   IF #command > 100 THEN
       "SandBoxData".MnualCommandMem := #command;
   END_IF;
   IF #command = 5000 THEN
       #data.Status.ToBp := true;
   END_IF;
   IF #command = 6000 THEN
       #data.Status.ToWp := true;
   END_IF;
   IF #command = 7000 THEN
       #data.Status.ToFp := true;
   END_IF;
END_REGION

REGION Network 3 (SCL): check new cylinder command
   //check if basic position req movement changed
   IF #data.Status.ToBp <> #dataOld.Status.ToBp AND #data.Status.ToBp THEN
       #data.Status.ToFp := false;
       #data.Status.ToWp := false;
       IF #noCollision THEN
           #data.Status.ToFp := false;
           #data.Status.ToWp := false;
       ELSE
           #data.Status.ToBp := false;
       END_IF;
   END_IF;
   //check if work position req movement changed
   IF #data.Status.ToWp <> #dataOld.Status.ToWp AND #data.Status.ToWp THEN
       IF #noCollision  THEN
           #data.Status.ToFp := false;
           #data.Status.ToBp := false;
       ELSE
           #data.Status.ToWp := false;
       END_IF;
   END_IF;
   //check if free position req movement changed
   IF #data.Status.ToFp <> #dataOld.Status.ToFp AND #data.Status.ToFp THEN
       #data.Status.ToBp := false;
       #data.Status.ToWp := false;
       IF #noCollision THEN
           #data.Status.ToBp := false;
           #data.Status.ToWp := false;
       ELSE
           #data.Status.ToFp := false;
       END_IF;
   END_IF;
   //store actual cylinder status to old
   #dataOld.Status := #data.Status;
END_REGION

REGION Network 4
   RUNG wire#powerrail
      Contact( #HydraulicActive )
      { S7_Templates := "time_type := Time" } #IEC_Timer_0_Instance.TON(pt := t#3s, et =>)
   END_RUNG
   // the same network as SCL:
   #IEC_Timer_0_Instance(IN := #HydraulicActive, PT := t#3s);   // TON
END_REGION

REGION Network 5: Start move to basic position
   RUNG wire#powerrail
      Contact( #data.Status.ToBp )
      Contact( #IEC_Timer_0_Instance.Q )
      Sub(in1 := 0.0, in2 := #data.FlowCmd, out => #data.Flow)
      Move(in := #data.PressureCmd, out1 => #data.Pressure)
   END_RUNG
   // the same network as SCL:
   IF #data.Status.ToBp AND #IEC_Timer_0_Instance.Q THEN
       #data.Flow := 0.0 - #data.FlowCmd;
       #data.Pressure := #data.PressureCmd;
   END_IF;
END_REGION

REGION Network 6: Start move to working position
   RUNG wire#powerrail
      Contact( #data.Status.ToWp )
      Contact( #IEC_Timer_0_Instance.Q )
      Move(in := #data.FlowCmd, out1 => #data.Flow)
      Move(in := #data.PressureCmd, out1 => #data.Pressure)
   END_RUNG
   // the same network as SCL:
   IF #data.Status.ToWp AND #IEC_Timer_0_Instance.Q THEN
       #data.Flow := #data.FlowCmd;
       #data.Pressure := #data.PressureCmd;
   END_IF;
END_REGION

REGION Network 7: Small movement to basic position when no command active and hydraulic running
   RUNG wire#powerrail
      Contact( #HydraulicActive )
      I_Contact( #data.Status.ToBp )
      I_Contact( #data.Status.ToWp )
      I_Contact( #data.Status.ToFp )
      { S7_Templates := "SrcType := Real" } LE_Contact(in1 := #data.Position, in2 := #BasicPositionMax)
      { S7_Templates := "SrcType := Real" } GE_Contact(in1 := #data.Position, in2 := #BasicPositionMin)
      Move(in := 3.0, out1 => #data.Pressure)
      Move(in := -5.0, out1 => #data.Flow)
   END_RUNG
   // the same network as SCL:
   IF #HydraulicActive AND NOT #data.Status.ToBp AND NOT #data.Status.ToWp AND NOT #data.Status.ToFp AND (#data.Position <= #BasicPositionMax) AND (#data.Position >= #BasicPositionMin) THEN
       #data.Pressure := 3.0;
       #data.Flow := -5.0;
   END_IF;
END_REGION

REGION Network 8: Stop movement when abou allowed position
   RUNG wire#powerrail
      { S7_Templates := "SrcType := Real" } GT_Contact(in1 := #data.Position, in2 := #MaxPosition)
      wire#w1
      I_Contact( #data.Status.ToBp )
      Contact( #HydraulicActive )
      Move(in := 3.0, out1 => #data.Pressure)
      Move(in := -5.0, out1 => #data.Flow)
   END_RUNG
   RUNG wire#w1
      I_Contact( #data.Status.ToBp )
      I_Contact( #HydraulicActive )
      Move(in := 0.0, out1 => #data.Pressure)
      Move(in := 0.0, out1 => #data.Flow)
   END_RUNG
   // the same network as SCL:
   #_w1 := #data.Position > #MaxPosition;
   IF #_w1 AND NOT #data.Status.ToBp AND #HydraulicActive THEN
       #data.Pressure := 3.0;
       #data.Flow := -5.0;
   END_IF;
   IF #_w1 AND NOT #data.Status.ToBp AND NOT #HydraulicActive THEN
       #data.Pressure := 0.0;
       #data.Flow := 0.0;
   END_IF;
END_REGION

REGION Network 9: In basic position
   RUNG wire#powerrail
      Contact( #data.Status.ToBp )
      wire#w1
      I_Contact( "FirstScan" )
      wire#w2
      Add(in1 := #BasicPositionMin, in2 := 1.0, out => #BasicPositionMin_1mm_margin)
      Add(in1 := #BasicPositionMax, in2 := -1.0, out => #BasicPositionMax_1mm_margin)
   END_RUNG
   RUNG wire#powerrail
      Contact( #data.Status.ToFp )
   END_RUNG wire#w1
   RUNG wire#w2
      { S7_Templates := "SrcType := Real" } GE_Contact(in1 := #data.Position, in2 := #BasicPositionMin)
      { S7_Templates := "SrcType := Real" } LE_Contact(in1 := #data.Position, in2 := #BasicPositionMax)
      { S7_Templates := "time_type := Time" } #IEC_Timer_0_Instance_1.TON(pt := t#50ms, et =>)
   END_RUNG
   RUNG wire#w2
      { S7_Templates := "SrcType := Real" } GE_Contact(in1 := #data.Position, in2 := #BasicPositionMin_1mm_margin)
      { S7_Templates := "SrcType := Real" } LE_Contact(in1 := #data.Position, in2 := #BasicPositionMax_1mm_margin)
      Coil( #data.InBp_1mm_margin )
   END_RUNG
   RUNG wire#w2
      Contact( #IEC_Timer_0_Instance_1.Q )
      wire#w3
      Coil( #data.Status.InBp )
   END_RUNG
   RUNG wire#w2
      Contact( #data.InBp_1mm_margin )
   END_RUNG wire#w3
   // the same network as SCL:
   #_w1 := (#data.Status.ToBp OR #data.Status.ToFp) AND NOT "FirstScan";
   IF #_w1 THEN
       #BasicPositionMin_1mm_margin := #BasicPositionMin + 1.0;
       #BasicPositionMax_1mm_margin := #BasicPositionMax + (-1.0);
   END_IF;
   #IEC_Timer_0_Instance_1(IN := #_w1 AND (#data.Position >= #BasicPositionMin) AND (#data.Position <= #BasicPositionMax),   // TON
                           PT := t#50ms);
   #data.InBp_1mm_margin := #_w1 AND (#data.Position >= #BasicPositionMin_1mm_margin) AND (#data.Position <= #BasicPositionMax_1mm_margin);
   #data.Status.InBp := #_w1 AND (#IEC_Timer_0_Instance_1.Q OR #data.InBp_1mm_margin);
END_REGION

REGION Network 10: Stand still - start stand still
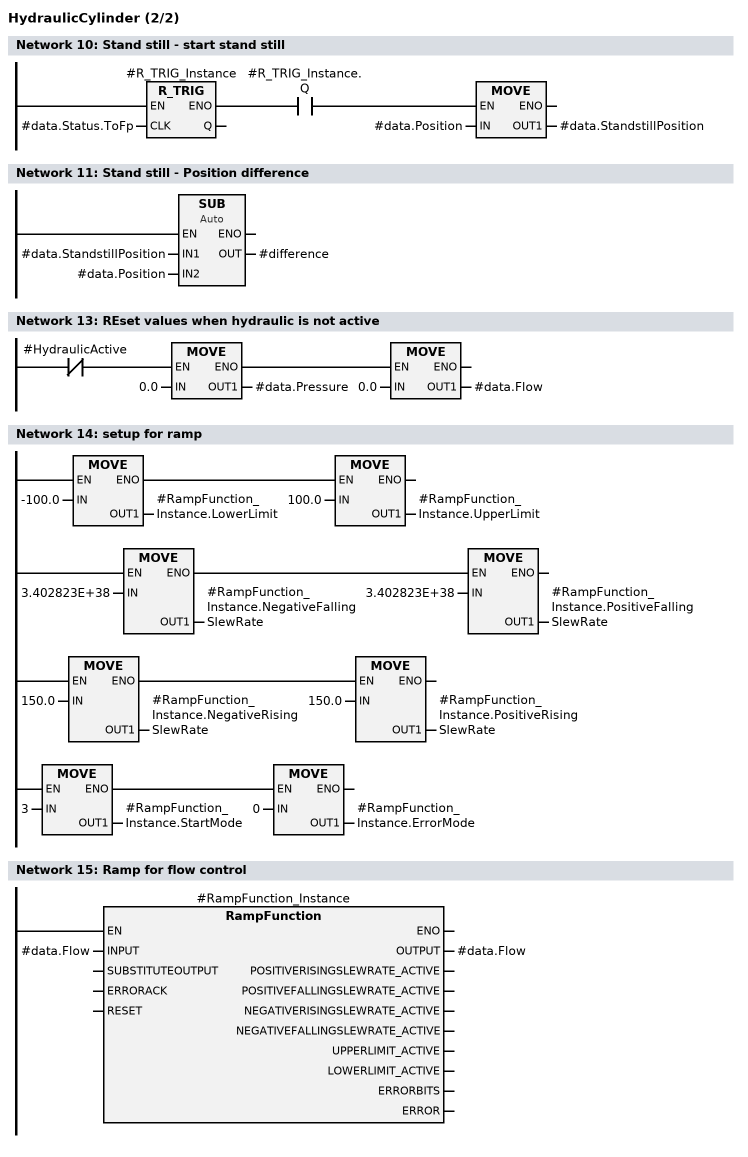
   RUNG wire#powerrail
      #R_TRIG_Instance.R_TRIG(CLK := #data.Status.ToFp, Q =>)
      Contact( #R_TRIG_Instance.Q )
      Move(in := #data.Position, out1 => #data.StandstillPosition)
   END_RUNG
   // the same network as SCL:
   #R_TRIG_Instance(CLK := #data.Status.ToFp, ENO => #_w1);   // R_TRIG
   IF #_w1 AND #R_TRIG_Instance.Q THEN #data.StandstillPosition := #data.Position; END_IF;
END_REGION

REGION Network 11: Stand still - Position difference
   RUNG wire#powerrail
      Sub(in1 := #data.StandstillPosition, in2 := #data.Position, out => #difference)
   END_RUNG
   // the same network as SCL:
   #difference := #data.StandstillPosition - #data.Position;
END_REGION

REGION Network 12 (SCL): Stand still - count regulation

   IF #data.Status.ToFp THEN
       #re := #difference;
       #re := #re * 10;
       IF #re > 0 THEN
           #re := #re + 5;
       END_IF;
       IF #re > 30 THEN
           #re := 30;
       END_IF;
       IF #re < -30 THEN
           #re := -30;
       END_IF;
       #data.Flow := #re;
       #data.Pressure := #data.PressureCmd;

       #data.Flow := 0;
       #data.Pressure := 0;

   END_IF;

   ;
END_REGION

REGION Network 13: REset values when hydraulic is not active
   RUNG wire#powerrail
      I_Contact( #HydraulicActive )
      Move(in := 0.0, out1 => #data.Pressure)
      Move(in := 0.0, out1 => #data.Flow)
   END_RUNG
   // the same network as SCL:
   IF NOT #HydraulicActive THEN
       #data.Pressure := 0.0;
       #data.Flow := 0.0;
   END_IF;
END_REGION

REGION Network 14: setup for ramp
   RUNG wire#powerrail
      Move(in := -100.0, out1 => #RampFunction_Instance.LowerLimit)
      Move(in := 100.0, out1 => #RampFunction_Instance.UpperLimit)
   END_RUNG
   RUNG wire#powerrail
      Move(in := 3.402823E+38, out1 => #RampFunction_Instance.NegativeFallingSlewRate)
      Move(in := 3.402823E+38, out1 => #RampFunction_Instance.PositiveFallingSlewRate)
   END_RUNG
   RUNG wire#powerrail
      Move(in := 150.0, out1 => #RampFunction_Instance.NegativeRisingSlewRate)
      Move(in := 150.0, out1 => #RampFunction_Instance.PositiveRisingSlewRate)
   END_RUNG
   RUNG wire#powerrail
      Move(in := 3, out1 => #RampFunction_Instance.StartMode)
      Move(in := 0, out1 => #RampFunction_Instance.ErrorMode)
   END_RUNG
   // the same network as SCL:
   #RampFunction_Instance.LowerLimit := -100.0;
   #RampFunction_Instance.UpperLimit := 100.0;
   #RampFunction_Instance.NegativeFallingSlewRate := 3.402823E+38;
   #RampFunction_Instance.PositiveFallingSlewRate := 3.402823E+38;
   #RampFunction_Instance.NegativeRisingSlewRate := 150.0;
   #RampFunction_Instance.PositiveRisingSlewRate := 150.0;
   #RampFunction_Instance.StartMode := 3;
   #RampFunction_Instance.ErrorMode := 0;
END_REGION

REGION Network 15: Ramp for flow control
   RUNG wire#powerrail
      #RampFunction_Instance.RampFunction(Input := #data.Flow, SubstituteOutput :=, ErrorAck :=, Reset :=, Output => #data.Flow, PositiveRisingSlewRate_Active =>, PositiveFallingSlewRate_Active =>, NegativeRisingSlewRate_Active =>, NegativeFallingSlewRate_Active =>, UpperLimit_Active =>, LowerLimit_Active =>, ErrorBits =>, Error =>)
   END_RUNG
   // the same network as SCL:
   #RampFunction_Instance(Input := #data.Flow, Output => #data.Flow);   // RampFunction
END_REGION
END_FUNCTION_BLOCK

FUNCTION_BLOCK "FittingCycle"   // FB35, LAD
{ S7_Optimized_Access := 'TRUE' }
VERSION : 0.1
// stored: AutoNumber true, IsIECCheckEnabled false, IsRetainMemResEnabled false, MemoryReserve 100, SetENOAutomatically false, UDAEnableTagReadback false
   VAR_INPUT
      parameters : "UDT_FittingParameters";
      basicPosition : Bool;
      MaxPosition : Real;
      endStopCylinderActive : Bool;
      shiftSupportToWork : Bool;
      rivetSensor : Bool;
      rivetStatusOtherCylinder : SInt;
   END_VAR
   VAR_IN_OUT
      HydraulicCylinder : "UDT_HydraulicCylinderData";
      dataFitting : "UDT_FittingStatus";
      dataDigiforce : "UDT_Digiforce";
      stopperForWedgeCylinder : "UDT_Cylinder";
      supportCylinder : "UDT_Cylinder";
      wedgeCylinder : "UDT_Cylinder";
      MeasuredData : "UDT_Results_Cupforming";
   END_VAR
   VAR
      cnt : Int;
      R_TRIG_Instance { S7_SetPoint := 'True'} : R_TRIG;
      H2Reached { S7_SetPoint := 'True'} : Bool;
      IEC_Timer_timeout { S7_SetPoint := 'True'} : TON_TIME;
      DigiforceStarted { S7_SetPoint := 'True'} : Bool;
      R_TRIG_Instance_1 { S7_SetPoint := 'True'} : R_TRIG;
      ton_WayWithTimeoutReached { S7_SetPoint := 'True'} : TON_TIME;
   END_VAR
   VAR_TEMP   // added for the SCL form of the ladder/FBD networks
      _w1 : Bool;
      _w2 : Bool;
   END_VAR
BEGIN

REGION Network 1: Check min max values
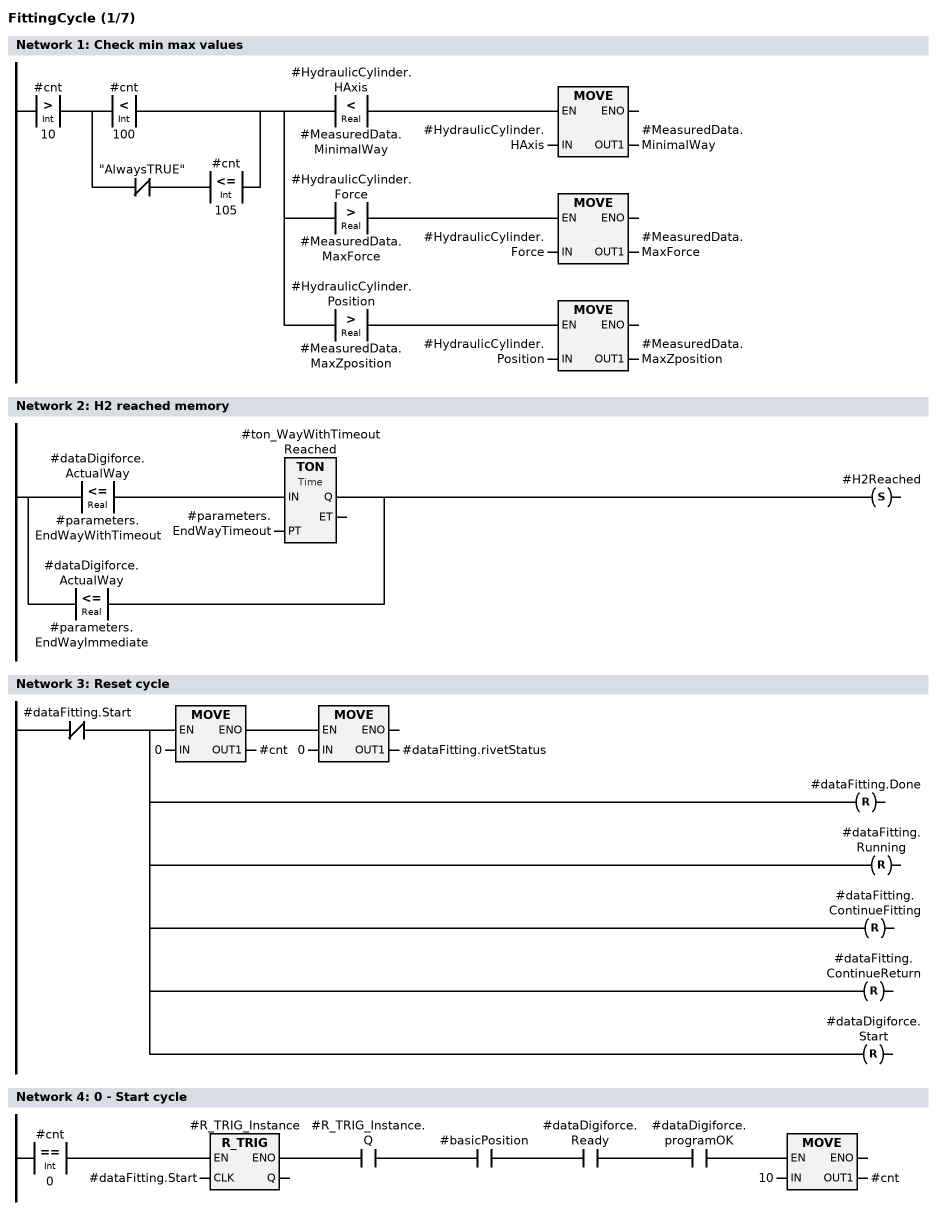
   RUNG wire#powerrail
      { S7_Templates := "SrcType := Int" } GT_Contact(in1 := #cnt, in2 := 10)
      wire#w1
      { S7_Templates := "SrcType := Int" } LT_Contact(in1 := #cnt, in2 := 100)
      wire#w2
      { S7_Templates := "SrcType := Real" } LT_Contact(in1 := #HydraulicCylinder.HAxis, in2 := #MeasuredData.MinimalWay)
      Move(in := #HydraulicCylinder.HAxis, out1 => #MeasuredData.MinimalWay)
   END_RUNG
   RUNG wire#w1
      I_Contact( "AlwaysTRUE" )
      { S7_Templates := "SrcType := Int" } LE_Contact(in1 := #cnt, in2 := 105)
   END_RUNG wire#w2
   RUNG wire#w2
      { S7_Templates := "SrcType := Real" } GT_Contact(in1 := #HydraulicCylinder.Force, in2 := #MeasuredData.MaxForce)
      Move(in := #HydraulicCylinder.Force, out1 => #MeasuredData.MaxForce)
   END_RUNG
   RUNG wire#w2
      { S7_Templates := "SrcType := Real" } GT_Contact(in1 := #HydraulicCylinder.Position, in2 := #MeasuredData.MaxZposition)
      Move(in := #HydraulicCylinder.Position, out1 => #MeasuredData.MaxZposition)
   END_RUNG
   // the same network as SCL:
   #_w1 := (#cnt > 10) AND ((#cnt < 100) OR (NOT "AlwaysTRUE" AND (#cnt <= 105)));
   IF #_w1 AND (#HydraulicCylinder.HAxis < #MeasuredData.MinimalWay) THEN
       #MeasuredData.MinimalWay := #HydraulicCylinder.HAxis;
   END_IF;
   IF #_w1 AND (#HydraulicCylinder.Force > #MeasuredData.MaxForce) THEN
       #MeasuredData.MaxForce := #HydraulicCylinder.Force;
   END_IF;
   IF #_w1 AND (#HydraulicCylinder.Position > #MeasuredData.MaxZposition) THEN
       #MeasuredData.MaxZposition := #HydraulicCylinder.Position;
   END_IF;
END_REGION

REGION Network 2: H2 reached memory
   RUNG wire#powerrail
      { S7_Templates := "SrcType := Real" } LE_Contact(in1 := #dataDigiforce.ActualWay, in2 := #parameters.EndWayWithTimeout)
      { S7_Templates := "time_type := Time" } #ton_WayWithTimeoutReached.TON(pt := #parameters.EndWayTimeout, et =>)
      wire#w1
      S_Coil( #H2Reached )
   END_RUNG
   RUNG wire#powerrail
      { S7_Templates := "SrcType := Real" } LE_Contact(in1 := #dataDigiforce.ActualWay, in2 := #parameters.EndWayImmediate)
   END_RUNG wire#w1
   // the same network as SCL:
   #ton_WayWithTimeoutReached(IN := #dataDigiforce.ActualWay <= #parameters.EndWayWithTimeout,   // TON
                           PT := #parameters.EndWayTimeout);
   IF #ton_WayWithTimeoutReached.Q OR (#dataDigiforce.ActualWay <= #parameters.EndWayImmediate) THEN
       #H2Reached := TRUE;
   END_IF;
END_REGION

REGION Network 3: Reset cycle
   RUNG wire#powerrail
      I_Contact( #dataFitting.Start )
      wire#w1
      Move(in := 0, out1 => #cnt)
      Move(in := 0, out1 => #dataFitting.rivetStatus)
   END_RUNG
   RUNG wire#w1
      R_Coil( #dataFitting.Done )
   END_RUNG
   RUNG wire#w1
      R_Coil( #dataFitting.Running )
   END_RUNG
   RUNG wire#w1
      R_Coil( #dataFitting.ContinueFitting )
   END_RUNG
   RUNG wire#w1
      R_Coil( #dataFitting.ContinueReturn )
   END_RUNG
   RUNG wire#w1
      R_Coil( #dataDigiforce.Start )
   END_RUNG
   // the same network as SCL:
   IF NOT #dataFitting.Start THEN
       #cnt := 0;
       #dataFitting.rivetStatus := 0;
       #dataFitting.Done := FALSE;
       #dataFitting.Running := FALSE;
       #dataFitting.ContinueFitting := FALSE;
       #dataFitting.ContinueReturn := FALSE;
       #dataDigiforce.Start := FALSE;
   END_IF;
END_REGION

REGION Network 4: 0 - Start cycle
   RUNG wire#powerrail
      { S7_Templates := "SrcType := Int" } EQ_Contact(in1 := #cnt, in2 := 0)
      #R_TRIG_Instance.R_TRIG(CLK := #dataFitting.Start, Q =>)
      Contact( #R_TRIG_Instance.Q )
      Contact( #basicPosition )
      Contact( #dataDigiforce.Ready )
      Contact( #dataDigiforce.programOK )
      Move(in := 10, out1 => #cnt)
   END_RUNG
   // the same network as SCL:
   #_w1 := #cnt = 0;
   #R_TRIG_Instance(EN := #_w1, CLK := #dataFitting.Start, ENO => #_w2);   // R_TRIG
   IF #_w2 AND #R_TRIG_Instance.Q AND #basicPosition AND #dataDigiforce.Ready AND #dataDigiforce.programOK THEN
       #cnt := 10;
   END_IF;
END_REGION

REGION Network 5: 10 - Start cycle
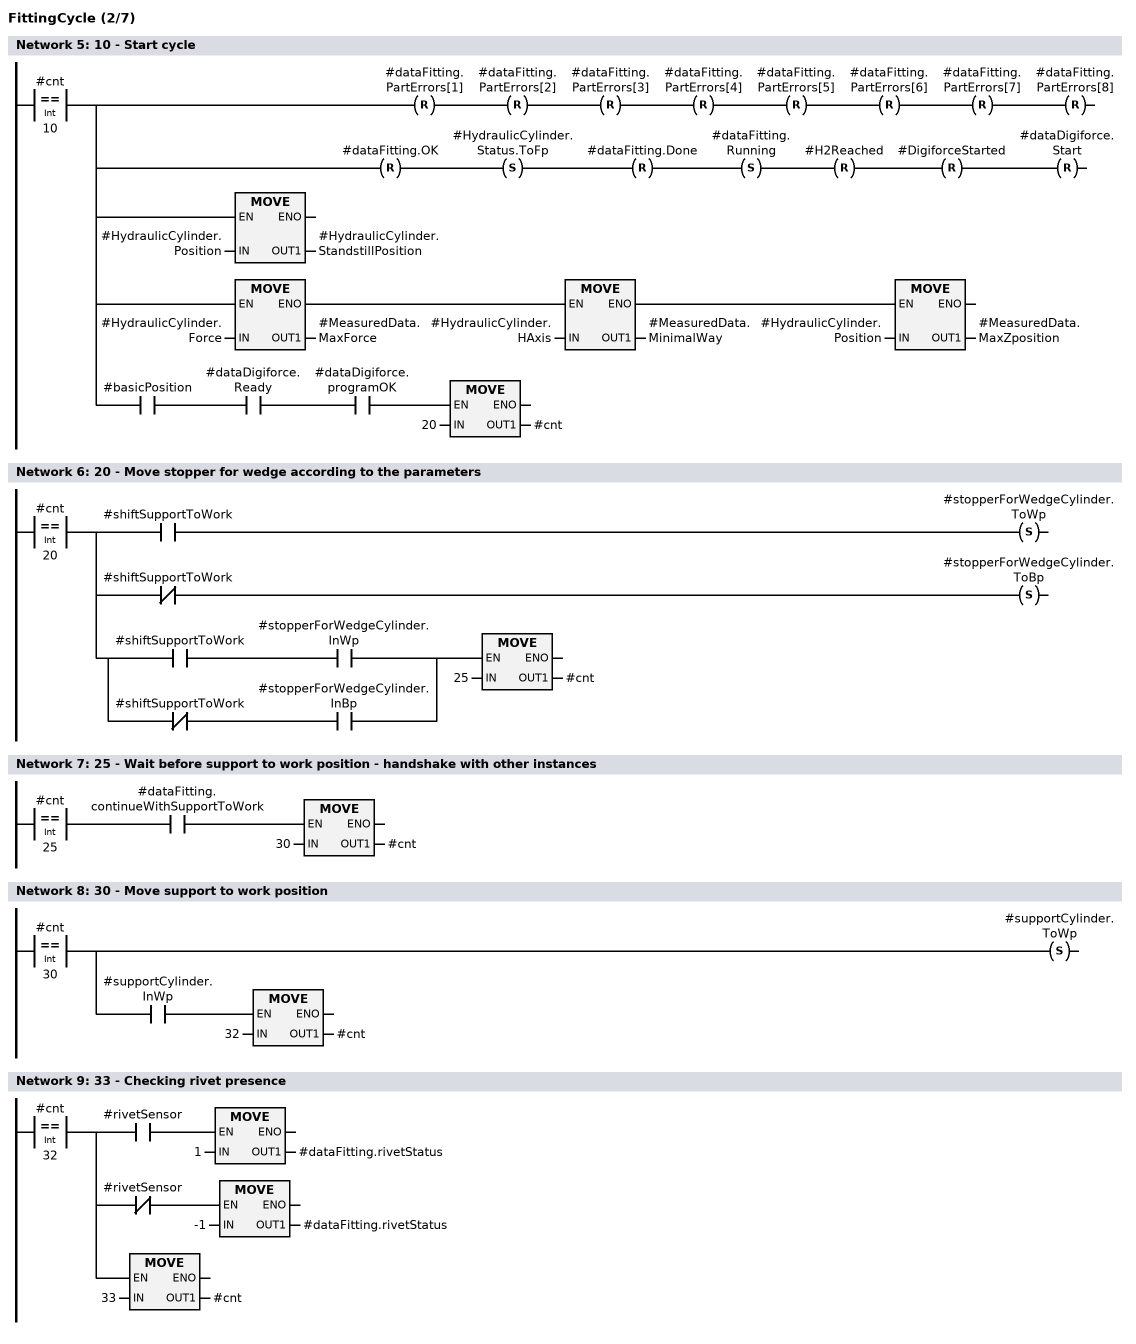
   RUNG wire#powerrail
      { S7_Templates := "SrcType := Int" } EQ_Contact(in1 := #cnt, in2 := 10)
      wire#w1
      R_Coil( #dataFitting.PartErrors[1] )
      R_Coil( #dataFitting.PartErrors[2] )
      R_Coil( #dataFitting.PartErrors[3] )
      R_Coil( #dataFitting.PartErrors[4] )
      R_Coil( #dataFitting.PartErrors[5] )
      R_Coil( #dataFitting.PartErrors[6] )
      R_Coil( #dataFitting.PartErrors[7] )
      R_Coil( #dataFitting.PartErrors[8] )
   END_RUNG
   RUNG wire#w1
      R_Coil( #dataFitting.OK )
      S_Coil( #HydraulicCylinder.Status.ToFp )
      R_Coil( #dataFitting.Done )
      S_Coil( #dataFitting.Running )
      R_Coil( #H2Reached )
      R_Coil( #DigiforceStarted )
      R_Coil( #dataDigiforce.Start )
   END_RUNG
   RUNG wire#w1
      Move(in := #HydraulicCylinder.Position, out1 => #HydraulicCylinder.StandstillPosition)
   END_RUNG
   RUNG wire#w1
      Move(in := #HydraulicCylinder.Force, out1 => #MeasuredData.MaxForce)
      Move(in := #HydraulicCylinder.HAxis, out1 => #MeasuredData.MinimalWay)
      Move(in := #HydraulicCylinder.Position, out1 => #MeasuredData.MaxZposition)
   END_RUNG
   RUNG wire#w1
      Contact( #basicPosition )
      Contact( #dataDigiforce.Ready )
      Contact( #dataDigiforce.programOK )
      Move(in := 20, out1 => #cnt)
   END_RUNG
   // the same network as SCL:
   #_w1 := #cnt = 10;
   IF #_w1 THEN
       #dataFitting.PartErrors[1] := FALSE;
       #dataFitting.PartErrors[2] := FALSE;
       #dataFitting.PartErrors[3] := FALSE;
       #dataFitting.PartErrors[4] := FALSE;
       #dataFitting.PartErrors[5] := FALSE;
       #dataFitting.PartErrors[6] := FALSE;
       #dataFitting.PartErrors[7] := FALSE;
       #dataFitting.PartErrors[8] := FALSE;
       #dataFitting.OK := FALSE;
       #HydraulicCylinder.Status.ToFp := TRUE;
       #dataFitting.Done := FALSE;
       #dataFitting.Running := TRUE;
       #H2Reached := FALSE;
       #DigiforceStarted := FALSE;
       #dataDigiforce.Start := FALSE;
       #HydraulicCylinder.StandstillPosition := #HydraulicCylinder.Position;
       #MeasuredData.MaxForce := #HydraulicCylinder.Force;
       #MeasuredData.MinimalWay := #HydraulicCylinder.HAxis;
       #MeasuredData.MaxZposition := #HydraulicCylinder.Position;
   END_IF;
   IF #_w1 AND #basicPosition AND #dataDigiforce.Ready AND #dataDigiforce.programOK THEN #cnt := 20; END_IF;
END_REGION

REGION Network 6: 20 - Move stopper for wedge according to the parameters
   RUNG wire#powerrail
      { S7_Templates := "SrcType := Int" } EQ_Contact(in1 := #cnt, in2 := 20)
      wire#w1
      Contact( #shiftSupportToWork )
      S_Coil( #stopperForWedgeCylinder.ToWp )
   END_RUNG
   RUNG wire#w1
      I_Contact( #shiftSupportToWork )
      S_Coil( #stopperForWedgeCylinder.ToBp )
   END_RUNG
   RUNG wire#w1
      Contact( #shiftSupportToWork )
      Contact( #stopperForWedgeCylinder.InWp )
      wire#w2
      Move(in := 25, out1 => #cnt)
   END_RUNG
   RUNG wire#w1
      I_Contact( #shiftSupportToWork )
      Contact( #stopperForWedgeCylinder.InBp )
   END_RUNG wire#w2
   // the same network as SCL:
   #_w1 := #cnt = 20;
   IF #_w1 AND #shiftSupportToWork THEN #stopperForWedgeCylinder.ToWp := TRUE; END_IF;
   IF #_w1 AND NOT #shiftSupportToWork THEN #stopperForWedgeCylinder.ToBp := TRUE; END_IF;
   IF #_w1 AND ((#shiftSupportToWork AND #stopperForWedgeCylinder.InWp) OR (NOT #shiftSupportToWork AND #stopperForWedgeCylinder.InBp)) THEN
       #cnt := 25;
   END_IF;
END_REGION

REGION Network 7: 25 - Wait before support to work position - handshake with other instances
   RUNG wire#powerrail
      { S7_Templates := "SrcType := Int" } EQ_Contact(in1 := #cnt, in2 := 25)
      Contact( #dataFitting.continueWithSupportToWork )
      Move(in := 30, out1 => #cnt)
   END_RUNG
   // the same network as SCL:
   IF (#cnt = 25) AND #dataFitting.continueWithSupportToWork THEN #cnt := 30; END_IF;
END_REGION

REGION Network 8: 30 - Move support to work position
   RUNG wire#powerrail
      { S7_Templates := "SrcType := Int" } EQ_Contact(in1 := #cnt, in2 := 30)
      wire#w1
      S_Coil( #supportCylinder.ToWp )
   END_RUNG
   RUNG wire#w1
      Contact( #supportCylinder.InWp )
      Move(in := 32, out1 => #cnt)
   END_RUNG
   // the same network as SCL:
   #_w1 := #cnt = 30;
   IF #_w1 THEN #supportCylinder.ToWp := TRUE; END_IF;
   IF #_w1 AND #supportCylinder.InWp THEN #cnt := 32; END_IF;
END_REGION

REGION Network 9: 33 - Checking rivet presence
   RUNG wire#powerrail
      { S7_Templates := "SrcType := Int" } EQ_Contact(in1 := #cnt, in2 := 32)
      wire#w1
      Contact( #rivetSensor )
      Move(in := 1, out1 => #dataFitting.rivetStatus)
   END_RUNG
   RUNG wire#w1
      I_Contact( #rivetSensor )
      Move(in := -1, out1 => #dataFitting.rivetStatus)
   END_RUNG
   RUNG wire#w1
      Move(in := 33, out1 => #cnt)
   END_RUNG
   // the same network as SCL:
   #_w1 := #cnt = 32;
   IF #_w1 AND #rivetSensor THEN #dataFitting.rivetStatus := 1; END_IF;
   IF #_w1 AND NOT #rivetSensor THEN #dataFitting.rivetStatus := -1; END_IF;
   IF #_w1 THEN #cnt := 33; END_IF;
END_REGION

REGION Network 10: 34 - Rivet presence result / handshake
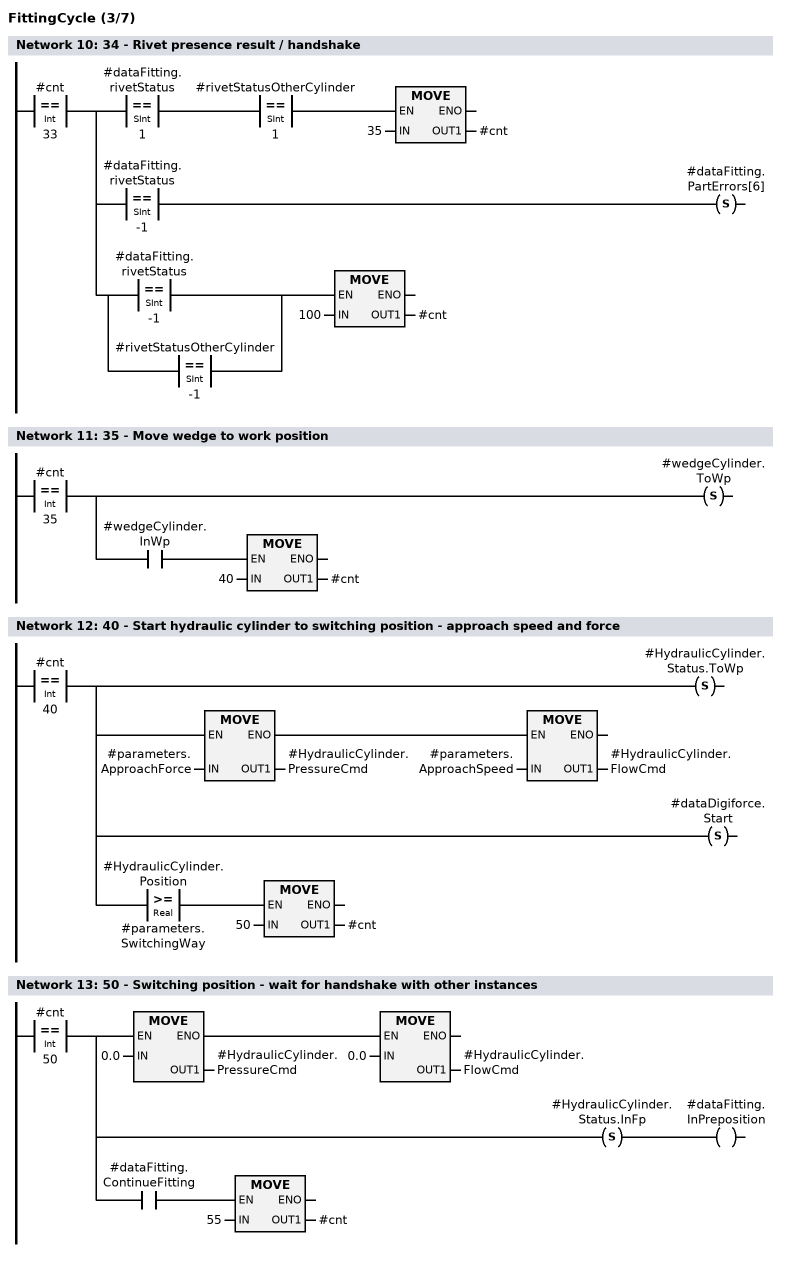
   RUNG wire#powerrail
      { S7_Templates := "SrcType := Int" } EQ_Contact(in1 := #cnt, in2 := 33)
      wire#w1
      { S7_Templates := "SrcType := SInt" } EQ_Contact(in1 := #dataFitting.rivetStatus, in2 := 1)
      { S7_Templates := "SrcType := SInt" } EQ_Contact(in1 := #rivetStatusOtherCylinder, in2 := 1)
      Move(in := 35, out1 => #cnt)
   END_RUNG
   RUNG wire#w1
      { S7_Templates := "SrcType := SInt" } EQ_Contact(in1 := #dataFitting.rivetStatus, in2 := -1)
      S_Coil( #dataFitting.PartErrors[6] )
   END_RUNG
   RUNG wire#w1
      { S7_Templates := "SrcType := SInt" } EQ_Contact(in1 := #dataFitting.rivetStatus, in2 := -1)
      wire#w2
      Move(in := 100, out1 => #cnt)
   END_RUNG
   RUNG wire#w1
      { S7_Templates := "SrcType := SInt" } EQ_Contact(in1 := #rivetStatusOtherCylinder, in2 := -1)
   END_RUNG wire#w2
   // the same network as SCL:
   #_w1 := #cnt = 33;
   IF #_w1 AND (#dataFitting.rivetStatus = 1) AND (#rivetStatusOtherCylinder = 1) THEN #cnt := 35; END_IF;
   IF #_w1 AND (#dataFitting.rivetStatus = (-1)) THEN #dataFitting.PartErrors[6] := TRUE; END_IF;
   IF #_w1 AND ((#dataFitting.rivetStatus = (-1)) OR (#rivetStatusOtherCylinder = (-1))) THEN
       #cnt := 100;
   END_IF;
END_REGION

REGION Network 11: 35 - Move wedge to work position
   RUNG wire#powerrail
      { S7_Templates := "SrcType := Int" } EQ_Contact(in1 := #cnt, in2 := 35)
      wire#w1
      S_Coil( #wedgeCylinder.ToWp )
   END_RUNG
   RUNG wire#w1
      Contact( #wedgeCylinder.InWp )
      Move(in := 40, out1 => #cnt)
   END_RUNG
   // the same network as SCL:
   #_w1 := #cnt = 35;
   IF #_w1 THEN #wedgeCylinder.ToWp := TRUE; END_IF;
   IF #_w1 AND #wedgeCylinder.InWp THEN #cnt := 40; END_IF;
END_REGION

REGION Network 12: 40 - Start hydraulic cylinder to switching position - approach speed and force
   RUNG wire#powerrail
      { S7_Templates := "SrcType := Int" } EQ_Contact(in1 := #cnt, in2 := 40)
      wire#w1
      S_Coil( #HydraulicCylinder.Status.ToWp )
   END_RUNG
   RUNG wire#w1
      Move(in := #parameters.ApproachForce, out1 => #HydraulicCylinder.PressureCmd)
      Move(in := #parameters.ApproachSpeed, out1 => #HydraulicCylinder.FlowCmd)
   END_RUNG
   RUNG wire#w1
      S_Coil( #dataDigiforce.Start )
   END_RUNG
   RUNG wire#w1
      { S7_Templates := "SrcType := Real" } GE_Contact(in1 := #HydraulicCylinder.Position, in2 := #parameters.SwitchingWay)
      Move(in := 50, out1 => #cnt)
   END_RUNG
   // the same network as SCL:
   #_w1 := #cnt = 40;
   IF #_w1 THEN
       #HydraulicCylinder.Status.ToWp := TRUE;
       #HydraulicCylinder.PressureCmd := #parameters.ApproachForce;
       #HydraulicCylinder.FlowCmd := #parameters.ApproachSpeed;
       #dataDigiforce.Start := TRUE;
   END_IF;
   IF #_w1 AND (#HydraulicCylinder.Position >= #parameters.SwitchingWay) THEN #cnt := 50; END_IF;
END_REGION

REGION Network 13: 50 - Switching position - wait for handshake with other instances
   RUNG wire#powerrail
      { S7_Templates := "SrcType := Int" } EQ_Contact(in1 := #cnt, in2 := 50)
      wire#w1
      Move(in := 0.0, out1 => #HydraulicCylinder.PressureCmd)
      Move(in := 0.0, out1 => #HydraulicCylinder.FlowCmd)
   END_RUNG
   RUNG wire#w1
      S_Coil( #HydraulicCylinder.Status.InFp )
      Coil( #dataFitting.InPreposition )
   END_RUNG
   RUNG wire#w1
      Contact( #dataFitting.ContinueFitting )
      Move(in := 55, out1 => #cnt)
   END_RUNG
   // the same network as SCL:
   #_w1 := #cnt = 50;
   IF #_w1 THEN
       #HydraulicCylinder.PressureCmd := 0.0;
       #HydraulicCylinder.FlowCmd := 0.0;
       #HydraulicCylinder.Status.InFp := TRUE;
   END_IF;
   #dataFitting.InPreposition := #_w1;
   IF #_w1 AND #dataFitting.ContinueFitting THEN #cnt := 55; END_IF;
END_REGION

REGION Network 14: 55 - Move sidemember to work position
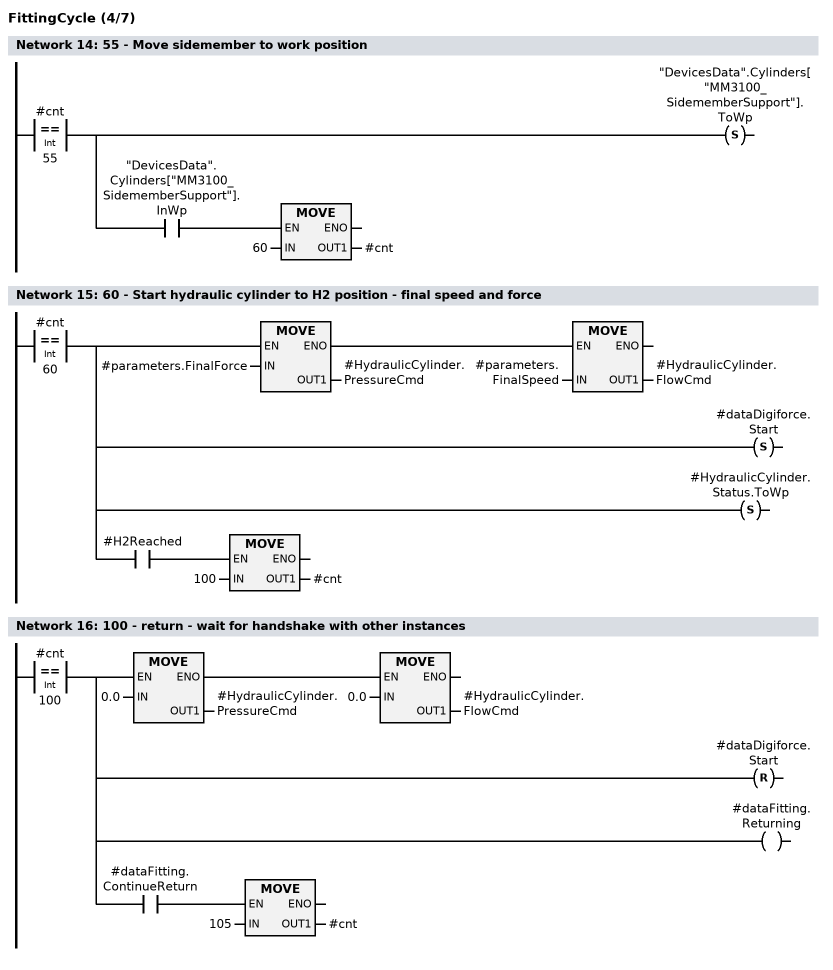
   RUNG wire#powerrail
      { S7_Templates := "SrcType := Int" } EQ_Contact(in1 := #cnt, in2 := 55)
      wire#w1
      S_Coil( "DevicesData".Cylinders["MM3100_SidememberSupport"].ToWp )
   END_RUNG
   RUNG wire#w1
      Contact( "DevicesData".Cylinders["MM3100_SidememberSupport"].InWp )
      Move(in := 60, out1 => #cnt)
   END_RUNG
   // the same network as SCL:
   #_w1 := #cnt = 55;
   IF #_w1 THEN "DevicesData".Cylinders["MM3100_SidememberSupport"].ToWp := TRUE; END_IF;
   IF #_w1 AND "DevicesData".Cylinders["MM3100_SidememberSupport"].InWp THEN #cnt := 60; END_IF;
END_REGION

REGION Network 15: 60 - Start hydraulic cylinder to H2 position - final speed and force
   RUNG wire#powerrail
      { S7_Templates := "SrcType := Int" } EQ_Contact(in1 := #cnt, in2 := 60)
      wire#w1
      Move(in := #parameters.FinalForce, out1 => #HydraulicCylinder.PressureCmd)
      Move(in := #parameters.FinalSpeed, out1 => #HydraulicCylinder.FlowCmd)
   END_RUNG
   RUNG wire#w1
      S_Coil( #dataDigiforce.Start )
   END_RUNG
   RUNG wire#w1
      S_Coil( #HydraulicCylinder.Status.ToWp )
   END_RUNG
   RUNG wire#w1
      Contact( #H2Reached )
      Move(in := 100, out1 => #cnt)
   END_RUNG
   // the same network as SCL:
   #_w1 := #cnt = 60;
   IF #_w1 THEN
       #HydraulicCylinder.PressureCmd := #parameters.FinalForce;
       #HydraulicCylinder.FlowCmd := #parameters.FinalSpeed;
       #dataDigiforce.Start := TRUE;
       #HydraulicCylinder.Status.ToWp := TRUE;
   END_IF;
   IF #_w1 AND #H2Reached THEN #cnt := 100; END_IF;
END_REGION

REGION Network 16: 100 - return - wait for handshake with other instances
   RUNG wire#powerrail
      { S7_Templates := "SrcType := Int" } EQ_Contact(in1 := #cnt, in2 := 100)
      wire#w1
      Move(in := 0.0, out1 => #HydraulicCylinder.PressureCmd)
      Move(in := 0.0, out1 => #HydraulicCylinder.FlowCmd)
   END_RUNG
   RUNG wire#w1
      R_Coil( #dataDigiforce.Start )
   END_RUNG
   RUNG wire#w1
      Coil( #dataFitting.Returning )
   END_RUNG
   RUNG wire#w1
      Contact( #dataFitting.ContinueReturn )
      Move(in := 105, out1 => #cnt)
   END_RUNG
   // the same network as SCL:
   #_w1 := #cnt = 100;
   IF #_w1 THEN
       #HydraulicCylinder.PressureCmd := 0.0;
       #HydraulicCylinder.FlowCmd := 0.0;
       #dataDigiforce.Start := FALSE;
   END_IF;
   #dataFitting.Returning := #_w1;
   IF #_w1 AND #dataFitting.ContinueReturn THEN #cnt := 105; END_IF;
END_REGION

REGION Network 17: 105 - Start returning
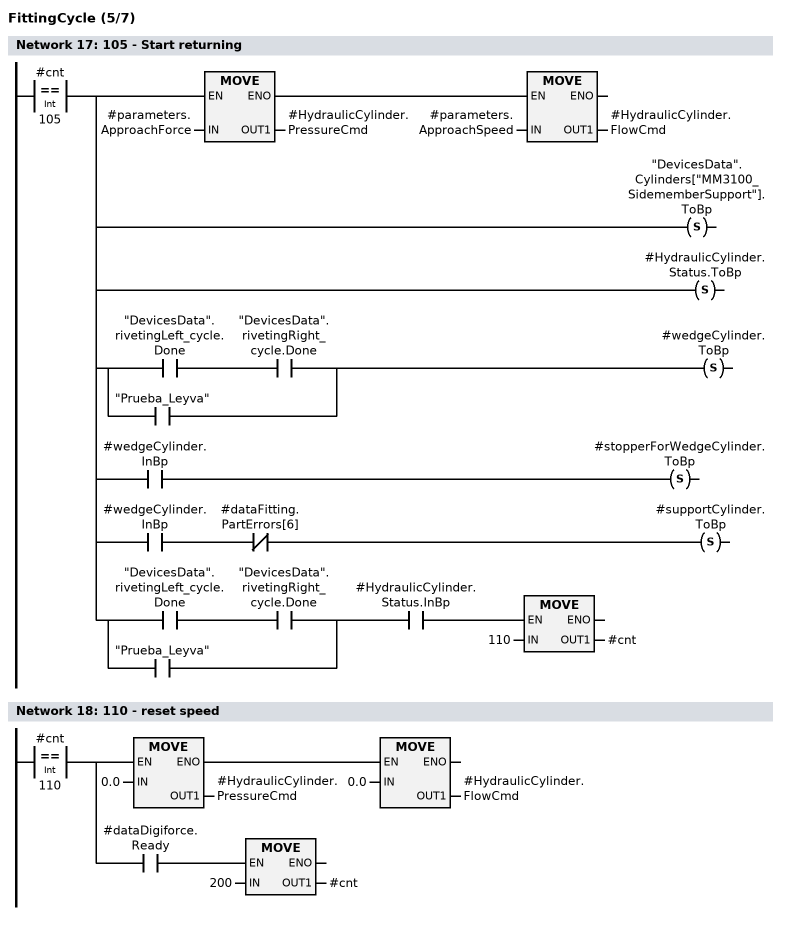
   RUNG wire#powerrail
      { S7_Templates := "SrcType := Int" } EQ_Contact(in1 := #cnt, in2 := 105)
      wire#w1
      Move(in := #parameters.ApproachForce, out1 => #HydraulicCylinder.PressureCmd)
      Move(in := #parameters.ApproachSpeed, out1 => #HydraulicCylinder.FlowCmd)
   END_RUNG
   RUNG wire#w1
      S_Coil( "DevicesData".Cylinders["MM3100_SidememberSupport"].ToBp )
   END_RUNG
   RUNG wire#w1
      S_Coil( #HydraulicCylinder.Status.ToBp )
   END_RUNG
   RUNG wire#w1
      Contact( "DevicesData".rivetingLeft_cycle.Done )
      Contact( "DevicesData".rivetingRight_cycle.Done )
      wire#w2
      S_Coil( #wedgeCylinder.ToBp )
   END_RUNG
   RUNG wire#w1
      Contact( "Prueba_Leyva" )
   END_RUNG wire#w2
   RUNG wire#w1
      Contact( #wedgeCylinder.InBp )
      S_Coil( #stopperForWedgeCylinder.ToBp )
   END_RUNG
   RUNG wire#w1
      Contact( #wedgeCylinder.InBp )
      I_Contact( #dataFitting.PartErrors[6] )
      S_Coil( #supportCylinder.ToBp )
   END_RUNG
   RUNG wire#w1
      Contact( "DevicesData".rivetingLeft_cycle.Done )
      Contact( "DevicesData".rivetingRight_cycle.Done )
      wire#w3
      Contact( #HydraulicCylinder.Status.InBp )
      Move(in := 110, out1 => #cnt)
   END_RUNG
   RUNG wire#w1
      Contact( "Prueba_Leyva" )
   END_RUNG wire#w3
   // the same network as SCL:
   #_w1 := #cnt = 105;
   IF #_w1 THEN
       #HydraulicCylinder.PressureCmd := #parameters.ApproachForce;
       #HydraulicCylinder.FlowCmd := #parameters.ApproachSpeed;
       "DevicesData".Cylinders["MM3100_SidememberSupport"].ToBp := TRUE;
       #HydraulicCylinder.Status.ToBp := TRUE;
   END_IF;
   IF #_w1 AND (("DevicesData".rivetingLeft_cycle.Done AND "DevicesData".rivetingRight_cycle.Done) OR "Prueba_Leyva") THEN
       #wedgeCylinder.ToBp := TRUE;
   END_IF;
   IF #_w1 AND #wedgeCylinder.InBp THEN #stopperForWedgeCylinder.ToBp := TRUE; END_IF;
   IF #_w1 AND #wedgeCylinder.InBp AND NOT #dataFitting.PartErrors[6] THEN
       #supportCylinder.ToBp := TRUE;
   END_IF;
   IF #_w1 AND (("DevicesData".rivetingLeft_cycle.Done AND "DevicesData".rivetingRight_cycle.Done) OR "Prueba_Leyva") AND #HydraulicCylinder.Status.InBp THEN
       #cnt := 110;
   END_IF;
END_REGION

REGION Network 18: 110 - reset speed
   RUNG wire#powerrail
      { S7_Templates := "SrcType := Int" } EQ_Contact(in1 := #cnt, in2 := 110)
      wire#w1
      Move(in := 0.0, out1 => #HydraulicCylinder.PressureCmd)
      Move(in := 0.0, out1 => #HydraulicCylinder.FlowCmd)
   END_RUNG
   RUNG wire#w1
      Contact( #dataDigiforce.Ready )
      Move(in := 200, out1 => #cnt)
   END_RUNG
   // the same network as SCL:
   #_w1 := #cnt = 110;
   IF #_w1 THEN
       #HydraulicCylinder.PressureCmd := 0.0;
       #HydraulicCylinder.FlowCmd := 0.0;
   END_IF;
   IF #_w1 AND #dataDigiforce.Ready THEN #cnt := 200; END_IF;
END_REGION

REGION Network 19: 200 - Move all cylinders to basic - evaluate result
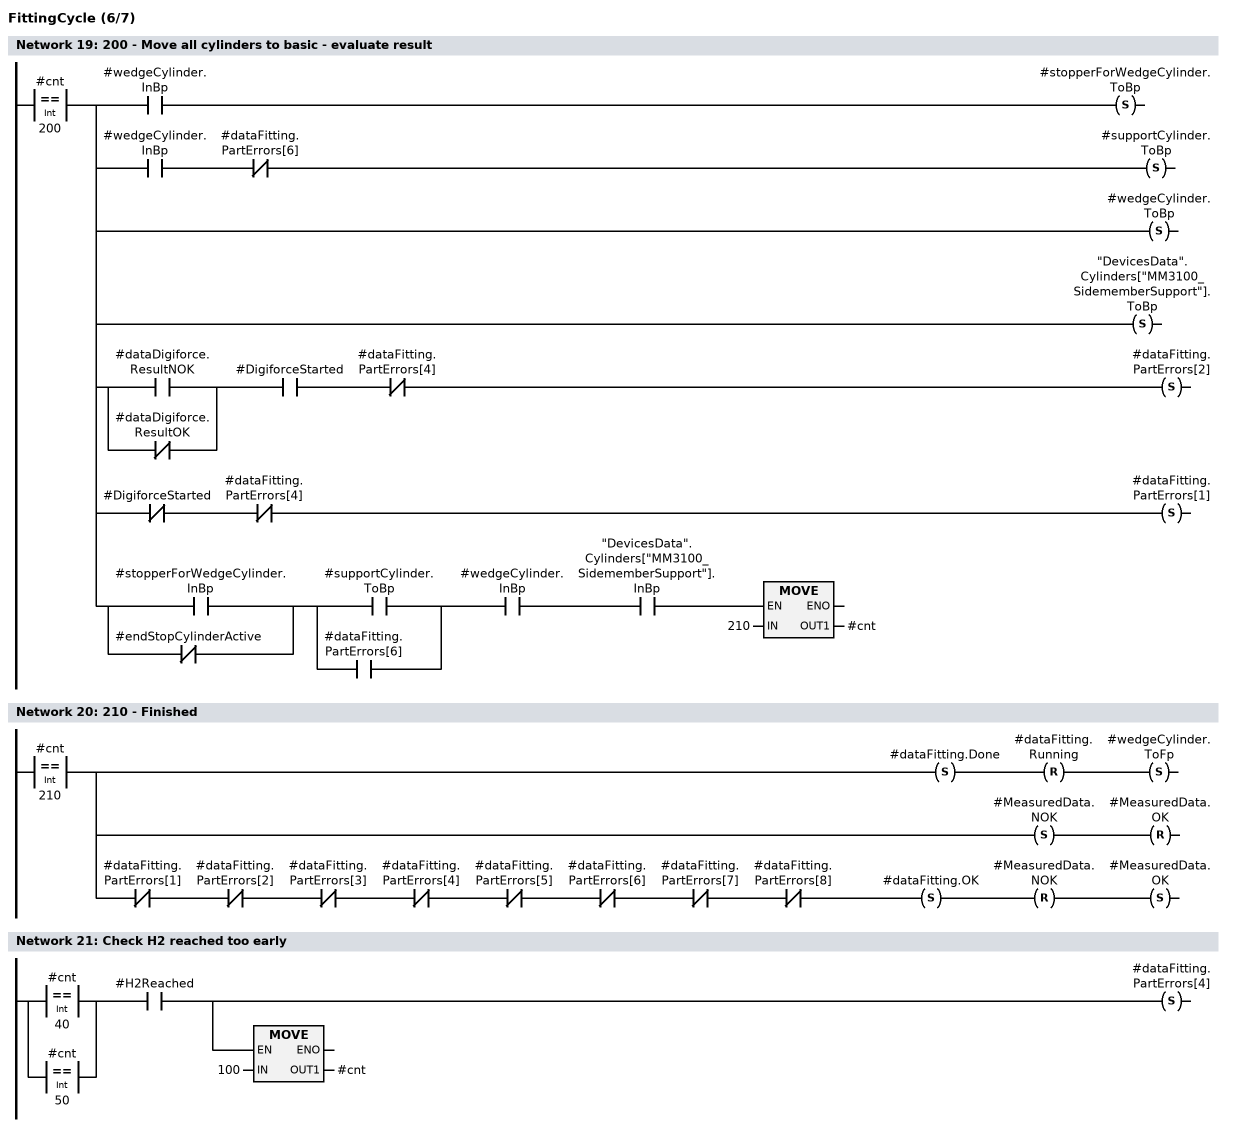
   RUNG wire#powerrail
      { S7_Templates := "SrcType := Int" } EQ_Contact(in1 := #cnt, in2 := 200)
      wire#w1
      Contact( #wedgeCylinder.InBp )
      S_Coil( #stopperForWedgeCylinder.ToBp )
   END_RUNG
   RUNG wire#w1
      Contact( #wedgeCylinder.InBp )
      I_Contact( #dataFitting.PartErrors[6] )
      S_Coil( #supportCylinder.ToBp )
   END_RUNG
   RUNG wire#w1
      S_Coil( #wedgeCylinder.ToBp )
   END_RUNG
   RUNG wire#w1
      S_Coil( "DevicesData".Cylinders["MM3100_SidememberSupport"].ToBp )
   END_RUNG
   RUNG wire#w1
      Contact( #dataDigiforce.ResultNOK )
      wire#w2
      Contact( #DigiforceStarted )
      I_Contact( #dataFitting.PartErrors[4] )
      S_Coil( #dataFitting.PartErrors[2] )
   END_RUNG
   RUNG wire#w1
      I_Contact( #dataDigiforce.ResultOK )
   END_RUNG wire#w2
   RUNG wire#w1
      I_Contact( #DigiforceStarted )
      I_Contact( #dataFitting.PartErrors[4] )
      S_Coil( #dataFitting.PartErrors[1] )
   END_RUNG
   RUNG wire#w1
      Contact( #stopperForWedgeCylinder.InBp )
      wire#w3
      Contact( #supportCylinder.ToBp )
      wire#w4
      Contact( #wedgeCylinder.InBp )
      Contact( "DevicesData".Cylinders["MM3100_SidememberSupport"].InBp )
      Move(in := 210, out1 => #cnt)
   END_RUNG
   RUNG wire#w1
      I_Contact( #endStopCylinderActive )
   END_RUNG wire#w3
   RUNG wire#w3
      Contact( #dataFitting.PartErrors[6] )
   END_RUNG wire#w4
   // the same network as SCL:
   #_w1 := #cnt = 200;
   IF #_w1 AND #wedgeCylinder.InBp THEN #stopperForWedgeCylinder.ToBp := TRUE; END_IF;
   IF #_w1 AND #wedgeCylinder.InBp AND NOT #dataFitting.PartErrors[6] THEN
       #supportCylinder.ToBp := TRUE;
   END_IF;
   IF #_w1 THEN
       #wedgeCylinder.ToBp := TRUE;
       "DevicesData".Cylinders["MM3100_SidememberSupport"].ToBp := TRUE;
   END_IF;
   IF #_w1 AND (#dataDigiforce.ResultNOK OR NOT #dataDigiforce.ResultOK) AND #DigiforceStarted AND NOT #dataFitting.PartErrors[4] THEN
       #dataFitting.PartErrors[2] := TRUE;
   END_IF;
   IF #_w1 AND NOT #DigiforceStarted AND NOT #dataFitting.PartErrors[4] THEN
       #dataFitting.PartErrors[1] := TRUE;
   END_IF;
   IF #_w1 AND (#stopperForWedgeCylinder.InBp OR NOT #endStopCylinderActive) AND (#supportCylinder.ToBp OR #dataFitting.PartErrors[6]) AND #wedgeCylinder.InBp AND "DevicesData".Cylinders["MM3100_SidememberSupport"].InBp THEN
       #cnt := 210;
   END_IF;
END_REGION

REGION Network 20: 210 - Finished
   RUNG wire#powerrail
      { S7_Templates := "SrcType := Int" } EQ_Contact(in1 := #cnt, in2 := 210)
      wire#w1
      S_Coil( #dataFitting.Done )
      R_Coil( #dataFitting.Running )
      S_Coil( #wedgeCylinder.ToFp )
   END_RUNG
   RUNG wire#w1
      S_Coil( #MeasuredData.NOK )
      R_Coil( #MeasuredData.OK )
   END_RUNG
   RUNG wire#w1
      I_Contact( #dataFitting.PartErrors[1] )
      I_Contact( #dataFitting.PartErrors[2] )
      I_Contact( #dataFitting.PartErrors[3] )
      I_Contact( #dataFitting.PartErrors[4] )
      I_Contact( #dataFitting.PartErrors[5] )
      I_Contact( #dataFitting.PartErrors[6] )
      I_Contact( #dataFitting.PartErrors[7] )
      I_Contact( #dataFitting.PartErrors[8] )
      S_Coil( #dataFitting.OK )
      R_Coil( #MeasuredData.NOK )
      S_Coil( #MeasuredData.OK )
   END_RUNG
   // the same network as SCL:
   #_w1 := #cnt = 210;
   IF #_w1 THEN
       #dataFitting.Done := TRUE;
       #dataFitting.Running := FALSE;
       #wedgeCylinder.ToFp := TRUE;
       #MeasuredData.NOK := TRUE;
       #MeasuredData.OK := FALSE;
   END_IF;
   IF #_w1 AND NOT #dataFitting.PartErrors[1] AND NOT #dataFitting.PartErrors[2] AND NOT #dataFitting.PartErrors[3] AND NOT #dataFitting.PartErrors[4] AND NOT #dataFitting.PartErrors[5] AND NOT #dataFitting.PartErrors[6] AND NOT #dataFitting.PartErrors[7] AND NOT #dataFitting.PartErrors[8] THEN
       #dataFitting.OK := TRUE;
       #MeasuredData.NOK := FALSE;
       #MeasuredData.OK := TRUE;
   END_IF;
END_REGION

REGION Network 21: Check H2 reached too early
   RUNG wire#powerrail
      { S7_Templates := "SrcType := Int" } EQ_Contact(in1 := #cnt, in2 := 40)
      wire#w1
      Contact( #H2Reached )
      wire#w2
      S_Coil( #dataFitting.PartErrors[4] )
   END_RUNG
   RUNG wire#powerrail
      { S7_Templates := "SrcType := Int" } EQ_Contact(in1 := #cnt, in2 := 50)
   END_RUNG wire#w1
   RUNG wire#w2
      Move(in := 100, out1 => #cnt)
   END_RUNG
   // the same network as SCL:
   IF ((#cnt = 40) OR (#cnt = 50)) AND #H2Reached THEN
       #dataFitting.PartErrors[4] := TRUE;
       #cnt := 100;
   END_IF;
END_REGION

REGION Network 22: Timeout
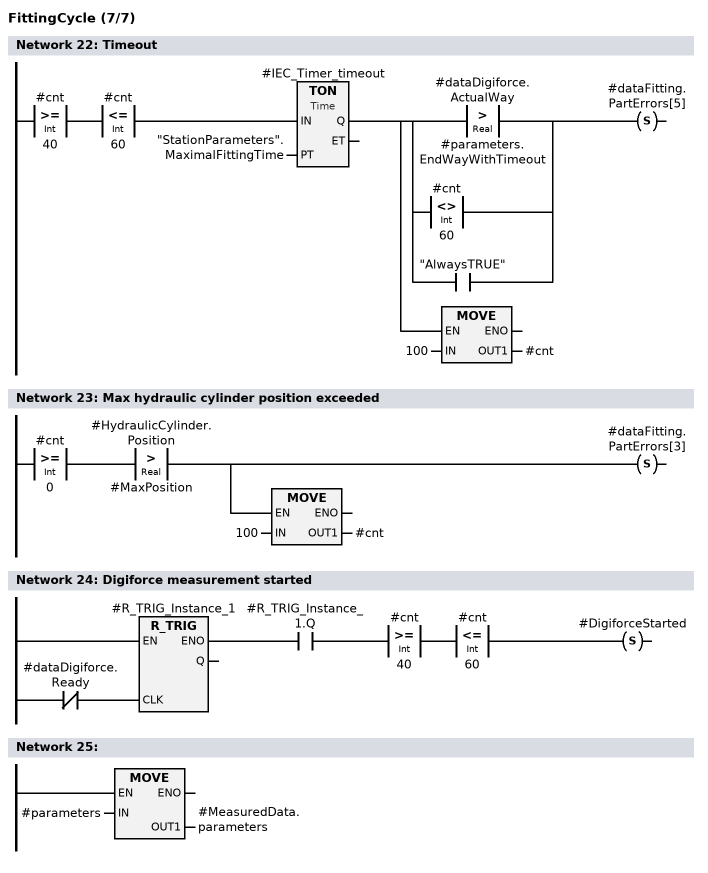
   RUNG wire#powerrail
      { S7_Templates := "SrcType := Int" } GE_Contact(in1 := #cnt, in2 := 40)
      { S7_Templates := "SrcType := Int" } LE_Contact(in1 := #cnt, in2 := 60)
      { S7_Templates := "time_type := Time" } #IEC_Timer_timeout.TON(pt := "StationParameters".MaximalFittingTime, et =>)
      wire#w1
      { S7_Templates := "SrcType := Real" } GT_Contact(in1 := #dataDigiforce.ActualWay, in2 := #parameters.EndWayWithTimeout)
      wire#w2
      S_Coil( #dataFitting.PartErrors[5] )
   END_RUNG
   RUNG wire#w1
      { S7_Templates := "SrcType := Int" } NE_Contact(in1 := #cnt, in2 := 60)
   END_RUNG wire#w2
   RUNG wire#w1
      Contact( "AlwaysTRUE" )
   END_RUNG wire#w2
   RUNG wire#w1
      Move(in := 100, out1 => #cnt)
   END_RUNG
   // the same network as SCL:
   #IEC_Timer_timeout(IN := (#cnt >= 40) AND (#cnt <= 60), PT := "StationParameters".MaximalFittingTime);   // TON
   IF #IEC_Timer_timeout.Q AND ((#dataDigiforce.ActualWay > #parameters.EndWayWithTimeout) OR (#cnt <> 60) OR "AlwaysTRUE") THEN
       #dataFitting.PartErrors[5] := TRUE;
   END_IF;
   IF #IEC_Timer_timeout.Q THEN #cnt := 100; END_IF;
END_REGION

REGION Network 23: Max hydraulic cylinder position exceeded
   RUNG wire#powerrail
      { S7_Templates := "SrcType := Int" } GE_Contact(in1 := #cnt, in2 := 0)
      { S7_Templates := "SrcType := Real" } GT_Contact(in1 := #HydraulicCylinder.Position, in2 := #MaxPosition)
      wire#w1
      S_Coil( #dataFitting.PartErrors[3] )
   END_RUNG
   RUNG wire#w1
      Move(in := 100, out1 => #cnt)
   END_RUNG
   // the same network as SCL:
   IF (#cnt >= 0) AND (#HydraulicCylinder.Position > #MaxPosition) THEN
       #dataFitting.PartErrors[3] := TRUE;
       #cnt := 100;
   END_IF;
END_REGION

REGION Network 24: Digiforce measurement started
   RUNG wire#powerrail
      #R_TRIG_Instance_1.R_TRIG(CLK := wire#w1, Q =>)
      Contact( #R_TRIG_Instance_1.Q )
      { S7_Templates := "SrcType := Int" } GE_Contact(in1 := #cnt, in2 := 40)
      { S7_Templates := "SrcType := Int" } LE_Contact(in1 := #cnt, in2 := 60)
      S_Coil( #DigiforceStarted )
   END_RUNG
   RUNG wire#powerrail
      I_Contact( #dataDigiforce.Ready )
   END_RUNG wire#w1
   // the same network as SCL:
   #R_TRIG_Instance_1(CLK := NOT #dataDigiforce.Ready, ENO => #_w1);   // R_TRIG
   IF #_w1 AND #R_TRIG_Instance_1.Q AND (#cnt >= 40) AND (#cnt <= 60) THEN #DigiforceStarted := TRUE; END_IF;
END_REGION

REGION Network 25
   RUNG wire#powerrail
      Move(in := #parameters, out1 => #MeasuredData.parameters)
   END_RUNG
   // the same network as SCL:
   #MeasuredData.parameters := #parameters;
END_REGION
END_FUNCTION_BLOCK

FUNCTION_BLOCK "HydraulicMotor"   // FB36, LAD
{ S7_Optimized_Access := 'TRUE' }
VERSION : 0.1
// stored: AutoNumber true, IsIECCheckEnabled false, IsRetainMemResEnabled false, MemoryReserve 100, SetENOAutomatically false, UDAEnableTagReadback false
   VAR_INPUT
      cycleActiveCupforming : Bool;
      cycleActiveRiveting : Bool;
      temp1nok : Bool;
      temp2nok : Bool;
   END_VAR
   VAR_IN_OUT
      data : "UDT_HydraulicPump";
      qKM20 : Bool;
      qMotor : Bool;
      qValveCupforming : Bool;
      qValveRiveting : Bool;
   END_VAR
   VAR
      R_TRIG_Instance { S7_SetPoint := 'True'} : R_TRIG;
      cnt { S7_SetPoint := 'True'} : Int;
      IEC_Timer_0_Instance { S7_SetPoint := 'True'} : TON_TIME;
      F_TRIG_Instance { S7_SetPoint := 'True'} : F_TRIG;
      IEC_Timer_0_Instance_1 { S7_SetPoint := 'True'} : TON_TIME;
   END_VAR
   VAR_TEMP   // added for the SCL form of the ladder/FBD networks
      _w1 : Bool;
   END_VAR
BEGIN

REGION Network 1: Start auto mode
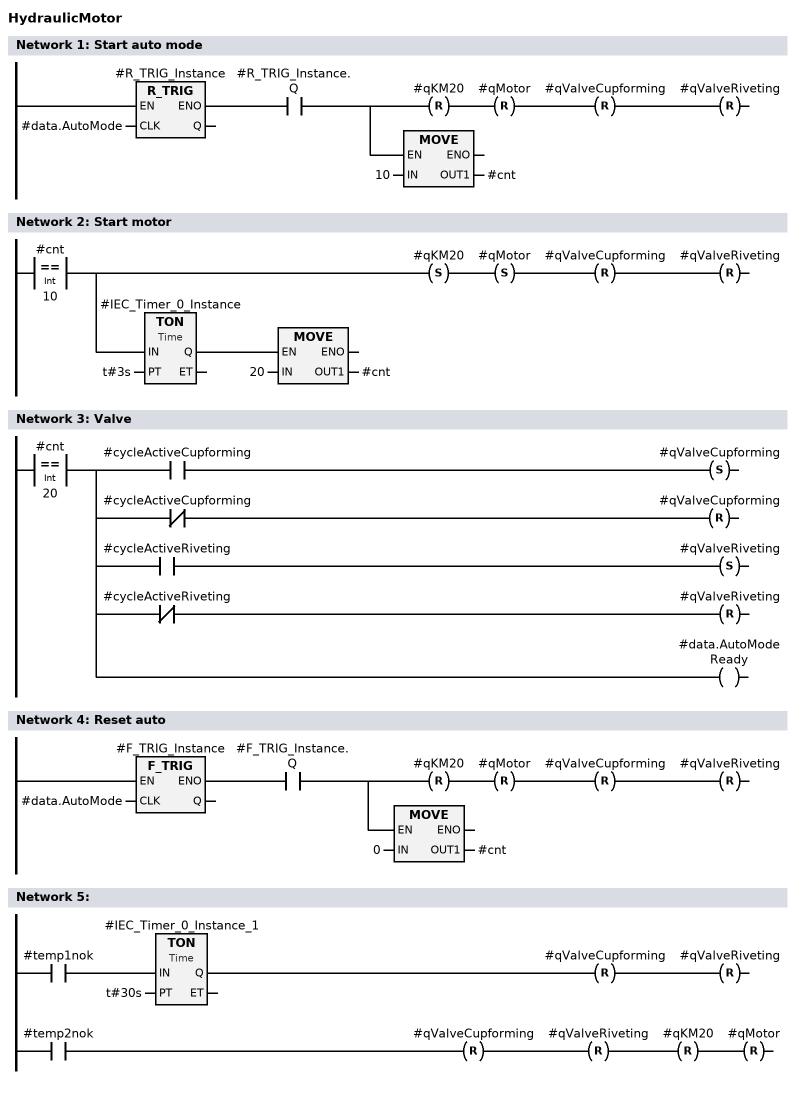
   RUNG wire#powerrail
      #R_TRIG_Instance.R_TRIG(CLK := #data.AutoMode, Q =>)
      Contact( #R_TRIG_Instance.Q )
      wire#w1
      R_Coil( #qKM20 )
      R_Coil( #qMotor )
      R_Coil( #qValveCupforming )
      R_Coil( #qValveRiveting )
   END_RUNG
   RUNG wire#w1
      Move(in := 10, out1 => #cnt)
   END_RUNG
   // the same network as SCL:
   #R_TRIG_Instance(CLK := #data.AutoMode, ENO => #_w1);   // R_TRIG
   IF #_w1 AND #R_TRIG_Instance.Q THEN
       #qKM20 := FALSE;
       #qMotor := FALSE;
       #qValveCupforming := FALSE;
       #qValveRiveting := FALSE;
       #cnt := 10;
   END_IF;
END_REGION

REGION Network 2: Start motor
   RUNG wire#powerrail
      { S7_Templates := "SrcType := Int" } EQ_Contact(in1 := #cnt, in2 := 10)
      wire#w1
      S_Coil( #qKM20 )
      S_Coil( #qMotor )
      R_Coil( #qValveCupforming )
      R_Coil( #qValveRiveting )
   END_RUNG
   RUNG wire#w1
      { S7_Templates := "time_type := Time" } #IEC_Timer_0_Instance.TON(pt := t#3s, et =>)
      Move(in := 20, out1 => #cnt)
   END_RUNG
   // the same network as SCL:
   #_w1 := #cnt = 10;
   IF #_w1 THEN
       #qKM20 := TRUE;
       #qMotor := TRUE;
       #qValveCupforming := FALSE;
       #qValveRiveting := FALSE;
   END_IF;
   #IEC_Timer_0_Instance(IN := #_w1, PT := t#3s);   // TON
   IF #IEC_Timer_0_Instance.Q THEN #cnt := 20; END_IF;
END_REGION

REGION Network 3: Valve
   RUNG wire#powerrail
      { S7_Templates := "SrcType := Int" } EQ_Contact(in1 := #cnt, in2 := 20)
      wire#w1
      Contact( #cycleActiveCupforming )
      S_Coil( #qValveCupforming )
   END_RUNG
   RUNG wire#w1
      I_Contact( #cycleActiveCupforming )
      R_Coil( #qValveCupforming )
   END_RUNG
   RUNG wire#w1
      Contact( #cycleActiveRiveting )
      S_Coil( #qValveRiveting )
   END_RUNG
   RUNG wire#w1
      I_Contact( #cycleActiveRiveting )
      R_Coil( #qValveRiveting )
   END_RUNG
   RUNG wire#w1
      Coil( #data.AutoModeReady )
   END_RUNG
   // the same network as SCL:
   #_w1 := #cnt = 20;
   IF #_w1 AND #cycleActiveCupforming THEN #qValveCupforming := TRUE; END_IF;
   IF #_w1 AND NOT #cycleActiveCupforming THEN #qValveCupforming := FALSE; END_IF;
   IF #_w1 AND #cycleActiveRiveting THEN #qValveRiveting := TRUE; END_IF;
   IF #_w1 AND NOT #cycleActiveRiveting THEN #qValveRiveting := FALSE; END_IF;
   #data.AutoModeReady := #_w1;
END_REGION

REGION Network 4: Reset auto
   RUNG wire#powerrail
      #F_TRIG_Instance.F_TRIG(CLK := #data.AutoMode, Q =>)
      Contact( #F_TRIG_Instance.Q )
      wire#w1
      R_Coil( #qKM20 )
      R_Coil( #qMotor )
      R_Coil( #qValveCupforming )
      R_Coil( #qValveRiveting )
   END_RUNG
   RUNG wire#w1
      Move(in := 0, out1 => #cnt)
   END_RUNG
   // the same network as SCL:
   #F_TRIG_Instance(CLK := #data.AutoMode, ENO => #_w1);   // F_TRIG
   IF #_w1 AND #F_TRIG_Instance.Q THEN
       #qKM20 := FALSE;
       #qMotor := FALSE;
       #qValveCupforming := FALSE;
       #qValveRiveting := FALSE;
       #cnt := 0;
   END_IF;
END_REGION

REGION Network 5
   RUNG wire#powerrail
      Contact( #temp1nok )
      { S7_Templates := "time_type := Time" } #IEC_Timer_0_Instance_1.TON(pt := t#30s, et =>)
      R_Coil( #qValveCupforming )
      R_Coil( #qValveRiveting )
   END_RUNG
   RUNG wire#powerrail
      Contact( #temp2nok )
      R_Coil( #qValveCupforming )
      R_Coil( #qValveRiveting )
      R_Coil( #qKM20 )
      R_Coil( #qMotor )
   END_RUNG
   // the same network as SCL:
   #IEC_Timer_0_Instance_1(IN := #temp1nok, PT := t#30s);   // TON
   IF #IEC_Timer_0_Instance_1.Q THEN
       #qValveCupforming := FALSE;
       #qValveRiveting := FALSE;
   END_IF;
   IF #temp2nok THEN
       #qValveCupforming := FALSE;
       #qValveRiveting := FALSE;
       #qKM20 := FALSE;
       #qMotor := FALSE;
   END_IF;
END_REGION
END_FUNCTION_BLOCK

FUNCTION_BLOCK "DiagnosticMain"
{ S7_Optimized_Access := 'TRUE' }
VERSION : 0.1
   VAR 
      i : Int;
      index : Int;
      state : Int;
   END_VAR


BEGIN
	//PN Device diagnostic
	"Devices_Diagnostic_DB"(PNIdentifier := "Local~PROFINET_IO-System");
	
	//IO Visualisation
	"IODiagnostic_DB"();
	
	
	
	//Make list of configured devices
	#index := 1;
	FOR #i := 1 TO 200 DO
	    IF "Devices_Diagnostic_DB".PNConfigured[#i] THEN
	        "DiagnosticConfigured".Adresses[#index] := #i;
	        #state := 0;
	        IF "Devices_Diagnostic_DB".PNFaulty[#i] THEN
	            #state := #state + w#16#0002;
	        END_IF;
	        IF "Devices_Diagnostic_DB".PNExist[#i] THEN
	            #state := #state + w#16#0001;
	        END_IF;
	        "DiagnosticConfigured".States[#index] := #state;
	        
	        "DiagnosticConfigured".Errors[#index] := "Devices_Diagnostic_DB".PNFaulty[#i];
	        "DiagnosticConfigured".Exists[#index] := "Devices_Diagnostic_DB".PNExist[#i];
	        #index := #index + 1;
	    END_IF;
	END_FOR;
	
	
	
	        
	
END_FUNCTION_BLOCK

FUNCTION_BLOCK "ScanCompare"
{ S7_Optimized_Access := 'TRUE' }
VERSION : 0.1
   VAR_INPUT 
      iDMC : String;
      iStringToCompare : String;
      iPosition : Int;
      iLength : Int;
   END_VAR

   VAR_OUTPUT 
      comparedString : String;
      OK : Bool;
   END_VAR


BEGIN
	#comparedString := MID(IN := #iDMC, L := #iLength, P := #iPosition);
	    
	#OK :=
	#comparedString = LEFT(IN := #iStringToCompare, L := #iLength);
	
END_FUNCTION_BLOCK

FUNCTION_BLOCK "ServoMain"
{ S7_Optimized_Access := 'TRUE' }
VERSION : 0.1
   VAR 
      "TO_BasicPos_TA1-3MA_Instance" {InstructionName := 'TO_BasicPos'; LibVersion := '1.0'} : TO_BasicPos;
      IEC_Timer_0_Instance {InstructionName := 'TON_TIME'; LibVersion := '1.0'} : TON_TIME;
      "ServoControl_TA1-3MA_Instance" : "ServoControl";
      IEC_Timer_0_Instance_1 {InstructionName := 'TP_TIME'; LibVersion := '1.0'} : TP_TIME;
   END_VAR


BEGIN
	
	
	IF "ModeSelection_DB".mode.activeMode <> "mode_1_manual" THEN
	    "DevicesData"."TA1-3MA".Jog1 := false;
	    "DevicesData"."TA1-3MA".Jog2 := false;
	END_IF;
	
	#IEC_Timer_0_Instance(IN := "DevicesData"."TA1-3MA".ExecuteMode AND "DevicesData"."TA1-3MA".ActMode = 2 AND NOT #IEC_Timer_0_Instance_1.Q,
	                      PT := t#100ms);
	#IEC_Timer_0_Instance_1(IN:=#IEC_Timer_0_Instance.Q,
	                        PT:=t#100ms);
	IF #IEC_Timer_0_Instance_1.Q THEN
	    "DevicesData"."TA1-3MA".ExecuteMode := FALSE;
	END_IF;
	
	#"ServoControl_TA1-3MA_Instance"(ServoParams := "StationParameters".Servo,
	                                 SafetyOK := "safety_signals"."4L+",
	                                 "Activate positioning" := FALSE,
	                                 ResetAlarm := "Alarms".Reset,
	                                 STOP := "safety_signals"."4L+" (*AND
	                                 "DevicesData".Cylinders["MM104_AutoejectGripperLifting"].InBp AND
	                                 "DevicesData".Cylinders["MM104_AutoejectGripperLifting"].ToBp*),
	                                 ConfigEPos_IO => "TO_TA1-3MA_DB".ConfigEPos,
	                                 ServoData := "DevicesData"."TA1-3MA");
	
	"TO_TA1-3MA_DB"(ModePos := "DevicesData"."TA1-3MA".ModePos,
	                EnableAxis := "DevicesData"."TA1-3MA".EnableAxis,
	                CancelTraversing := "DevicesData"."TA1-3MA".CancelTraversing,
	                IntermediateStop := "DevicesData"."TA1-3MA".IntermediateStop,
	                Positive := "DevicesData"."TA1-3MA".Positive,
	                Negative := "DevicesData"."TA1-3MA".Negative,
	                Jog1 := "DevicesData"."TA1-3MA".Jog1 AND
	                "DevicesData".Cylinders["MM104_AutoejectGripperLifting"].InBp AND
	                "DevicesData".Cylinders["MM104_AutoejectGripperLifting"].ToBp,
	                Jog2 := "DevicesData"."TA1-3MA".Jog2 AND
	                "DevicesData".Cylinders["MM104_AutoejectGripperLifting"].InBp AND
	                "DevicesData".Cylinders["MM104_AutoejectGripperLifting"].ToBp,
	                FlyRef := "DevicesData"."TA1-3MA".FlyRef,
	                AckError := "DevicesData"."TA1-3MA".AckError,
	                ExecuteMode := "DevicesData"."TA1-3MA".ExecuteMode AND
	                "DevicesData".Cylinders["MM104_AutoejectGripperLifting"].InBp AND
	                "DevicesData".Cylinders["MM104_AutoejectGripperLifting"].ToBp,
	                Position := "DevicesData"."TA1-3MA".Position,
	                Velocity := "DevicesData"."TA1-3MA".Velocity,
	                OverV := "DevicesData"."TA1-3MA".OverV,
	                OverAcc := "DevicesData"."TA1-3MA".OverAcc,
	                OverDec := "DevicesData"."TA1-3MA".OverDec,
	                //                      ConfigEPos:=_dword_in_,
	                AxisEnabled => "DevicesData"."TA1-3MA".AxisEnabled,
	                AxisPosOk => "DevicesData"."TA1-3MA".AxisPosOk,
	                AxisSpFixed => "DevicesData"."TA1-3MA".AxisSpFixed,
	                AxisRef => "DevicesData"."TA1-3MA".AxisRef,
	                AxisWarn => "DevicesData"."TA1-3MA".AxisWarn,
	                AxisError => "DevicesData"."TA1-3MA".AxisError,
	                Lockout => "DevicesData"."TA1-3MA".Lockout,
	 //               ActVelocity => "DevicesData"."TA1-3MA".ActVelocity,
	                ActPosition => "DevicesData"."TA1-3MA".ActPosition,
	                ActMode => "DevicesData"."TA1-3MA".ActMode,
	                EPosZSW1 => "DevicesData"."TA1-3MA".EPosZSW1,
	                EPosZSW2 => "DevicesData"."TA1-3MA".EPosZSW2,
	                ActWarn => "DevicesData"."TA1-3MA".ActWarn,
	                ActFault => "DevicesData"."TA1-3MA".ActFault,
	                Error => "DevicesData"."TA1-3MA".Error,
	                Status => "DevicesData"."TA1-3MA".Status,
	                DiagId => "DevicesData"."TA1-3MA".DiagID);
	
	"DevicesData"."TA1-3MA".ActVelocity := "TO_TA1-3MA_DB".ActVelocity / 220000;
	
	REGION zones
	    "DevicesData"."TA1-3MA".data.zones.inNOKpos := "DevicesData"."TA1-3MA".AxisRef AND "DevicesData"."TA1-3MA".AxisPosOk AND
	    "DevicesData"."TA1-3MA".ActPosition >= "StationParameters".ServoPositions[0] - 100 AND
	    "DevicesData"."TA1-3MA".ActPosition <= "StationParameters".ServoPositions[0] + 100;
	    
	    "DevicesData"."TA1-3MA".data.zones.inOKpos := "DevicesData"."TA1-3MA".AxisRef AND "DevicesData"."TA1-3MA".AxisPosOk AND
	    "DevicesData"."TA1-3MA".ActPosition >= "StationParameters".ServoPositions[1] - 100 AND
	    "DevicesData"."TA1-3MA".ActPosition <= "StationParameters".ServoPositions[1] + 100;
	    
	    "DevicesData"."TA1-3MA".data.zones.inST3jig := "DevicesData"."TA1-3MA".AxisRef AND "DevicesData"."TA1-3MA".AxisPosOk AND
	    "DevicesData"."TA1-3MA".ActPosition >= "StationParameters".ServoPositions[2] - 100 AND
	    "DevicesData"."TA1-3MA".ActPosition <= "StationParameters".ServoPositions[2] + 100;
	    
	    "DevicesData"."TA1-3MA".data.zones.outOfOKposZone := "DevicesData"."TA1-3MA".AxisRef AND
	    "DevicesData"."TA1-3MA".ActPosition <= "StationParameters".ServoPositions[0] + 10000 AND
	    "DevicesData"."TA1-3MA".Position <= "StationParameters".ServoPositions[0] + 100;
	    
	    "DevicesData"."TA1-3MA".data.zones.outOfST3zone := "DevicesData"."TA1-3MA".AxisRef AND
	    "DevicesData"."TA1-3MA".ActPosition <= "StationParameters".ServoPositions[1] + 10000 AND
	    "DevicesData"."TA1-3MA".Position <= "StationParameters".ServoPositions[1] + 100;
	END_REGION
	
	IF "ModeSelection_DB".mode.modeChanged THEN
	    "DevicesData"."TA1-3MA".EnableAxis := FALSE;
	END_IF;
	
	IF "ModeSelection_DB".mode.activeMode = "mode_2_base"
	    OR "ModeSelection_DB".mode.activeMode = "mode_3_automat" OR
	    "ModeSelection_DB".mode.activeMode = "mode_1_manual"
	THEN
	    "DevicesData"."TA1-3MA".EnableAxis :=
	    "DevicesData"."TA1-3MA".AxisEnabled
	    OR
	    NOT "DevicesData"."TA1-3MA".AxisEnabled AND
	    "Clock_1Hz";
	END_IF;
	
	
	
	
	
END_FUNCTION_BLOCK

FUNCTION_BLOCK "ServoControl"
{ S7_Optimized_Access := 'FALSE' }
VERSION : 0.1
   VAR_INPUT 
      ServoParams { ExternalAccessible := 'False'; ExternalVisible := 'False'; ExternalWritable := 'False'} : "UDT_ServoPrameters";
      SafetyOK { ExternalAccessible := 'False'; ExternalVisible := 'False'; ExternalWritable := 'False'} : Bool;
      "Activate positioning" : Bool;
      ResetAlarm { ExternalAccessible := 'False'; ExternalVisible := 'False'; ExternalWritable := 'False'} : Bool;
      STOP : Bool;
   END_VAR

   VAR_OUTPUT 
      ConfigEPos_IO : DWord;
   END_VAR

   VAR_IN_OUT 
      ServoData : "UDT_Servo";
   END_VAR

   VAR 
      IEC_Timer_0_Instance {InstructionName := 'TON_TIME'; LibVersion := '1.0'} : TON_TIME;
      R_TRIG_Instance {InstructionName := 'R_TRIG'; LibVersion := '1.0'} : R_TRIG;
      ConfigEPos_bits : "UDT_ConfigEPos";
      ConfigEPos_word { ExternalAccessible := 'False'; ExternalVisible := 'False'; ExternalWritable := 'False'} AT ConfigEPos_bits : DWord;
      IEC_Timer_0_Instance_1 {InstructionName := 'TON_TIME'; LibVersion := '1.0'} : TON_TIME;
   END_VAR


BEGIN
	//Copy parameter
	IF "ModeSelection_DB".mode.activeMode = "mode_2_base" OR "ModeSelection_DB".mode.activeMode = "mode_3_automat" OR "ModeSelection_DB".mode.activeMode = "mode_4_semiautomat" THEN
	    #ServoData.OverAcc := #ServoParams.OverAcc;
	    #ServoData.OverDec := #ServoParams.OverDec;
	    #ServoData.OverV := #ServoParams.OverV;
	    #ServoData.Velocity := #ServoParams.Velocity;
	END_IF;
	
	REGION configEPos
	    #ConfigEPos_bits.Off2 := TRUE;
	    #ConfigEPos_bits.Off3 := #STOP;
	    #ConfigEPos_bits.swLimitUsed := TRUE;
	    #ConfigEPos_bits.hwLimitUsed := TRUE;
	    #ConfigEPos_bits.reserve1 := FALSE;
	    #ConfigEPos_bits.reserve2 := FALSE;
	    #ConfigEPos_bits.reserve3 := FALSE;
	    #ConfigEPos_bits.reserve4 := FALSE;
	    #ConfigEPos_bits.reserve5 := FALSE;
	    #ConfigEPos_bits.reserve6 := FALSE;
	    #ConfigEPos_bits.reserve7 := FALSE;
	    #ConfigEPos_bits.reserve8 := FALSE;
	    #ConfigEPos_bits.reserve9 := FALSE;
	    #ConfigEPos_bits.reserve10 := FALSE;
	    #ConfigEPos_bits.reserve11 := FALSE;
	    #ConfigEPos_bits.reserve12 := FALSE;
	    #ConfigEPos_bits.reserve13 := FALSE;
	    #ConfigEPos_bits.reserve14 := FALSE;
	    #ConfigEPos_bits.reserve15 := FALSE;
	    #ConfigEPos_bits.reserve16 := FALSE;
	    #ConfigEPos_bits.reserve17 := FALSE;
	    #ConfigEPos_bits.reserve18 := FALSE;
	    #ConfigEPos_bits.reserve19 := FALSE;
	    #ConfigEPos_bits.reserve20 := FALSE;
	    #ConfigEPos_bits.reserve21 := FALSE;
	    #ConfigEPos_bits.reserve22 := FALSE;
	    #ConfigEPos_bits.reserve23 := FALSE;
	    #ConfigEPos_bits.reserve24 := FALSE;
	    #ConfigEPos_bits.reserve25 := FALSE;
	    #ConfigEPos_bits.reserve26 := FALSE;
	    #ConfigEPos_bits.reserve27 := FALSE;
	    #ConfigEPos_bits.reserve28 := FALSE;
	END_REGION
	
	//Enable movement
	#ServoData.CancelTraversing := #SafetyOK AND
	"DevicesData".Cylinders["MM104_AutoejectGripperLifting"].InBp AND
	"DevicesData".Cylinders["MM104_AutoejectGripperLifting"].ToBp;
	#ServoData.IntermediateStop := #SafetyOK;
	
	//Reset alarm
	#IEC_Timer_0_Instance_1(IN:=#ServoData.AckError,
	                        PT:=t#500ms);
	IF #IEC_Timer_0_Instance_1.Q THEN
	    #ServoData.AckError := FALSE;
	END_IF;
	IF #ResetAlarm AND (#ServoData.AxisError OR #ServoData.AxisWarn OR TRUE) THEN
	    #ServoData.AckError := true;
	END_IF;
	
	//Activate jog
	IF #ServoData.Jog1 OR #ServoData.Jog2 THEN
	    #ServoData.ModePos := 7;
	END_IF;
	
	//Activate positioning
	IF #"Activate positioning" THEN
	    #ServoData.ModePos := 2;
	END_IF;
	
	#ConfigEPos_IO := SWAP(#ConfigEPos_word);
	
	
END_FUNCTION_BLOCK

FUNCTION_BLOCK "RivetingCycle"   // FB52, LAD
{ S7_Optimized_Access := 'TRUE' }
VERSION : 0.1
// stored: AutoNumber true, IsIECCheckEnabled false, IsRetainMemResEnabled false, MemoryReserve 100, SetENOAutomatically false, UDAEnableTagReadback false
   VAR_INPUT
      parameters : Array[0..2] of USInt;
      basicPosition : Bool;
      twoRivets : Bool;
   END_VAR
   VAR_OUTPUT
      MeasuredData1 { ExternalAccessible := 'False'; ExternalVisible := 'False'; ExternalWritable := 'False'} : "UDT_Friedrich";
      MeasuredData2 { ExternalAccessible := 'False'; ExternalVisible := 'False'; ExternalWritable := 'False'} : "UDT_Friedrich";
   END_VAR
   VAR_IN_OUT
      riveter : "UDT_Friedrich";
      data : "UDT_FittingStatus";
      cylinderSupport : "UDT_Cylinder";
      cylinderShift : "UDT_Cylinder";
   END_VAR
   VAR
      cnt : Int;
      R_TRIG_Instance { S7_SetPoint := 'True'} : R_TRIG;
      IEC_Timer_timeout { S7_SetPoint := 'True'} : TON_TIME;
      R_TRIG_Instance_1 { S7_SetPoint := 'True'} : R_TRIG;
      ton_WayWithTimeoutReached { S7_SetPoint := 'True'} : TON_TIME;
   END_VAR
   VAR_TEMP   // added for the SCL form of the ladder/FBD networks
      _w1 : Bool;
      _w2 : Bool;
   END_VAR
BEGIN

REGION Network 1: Reset cycle
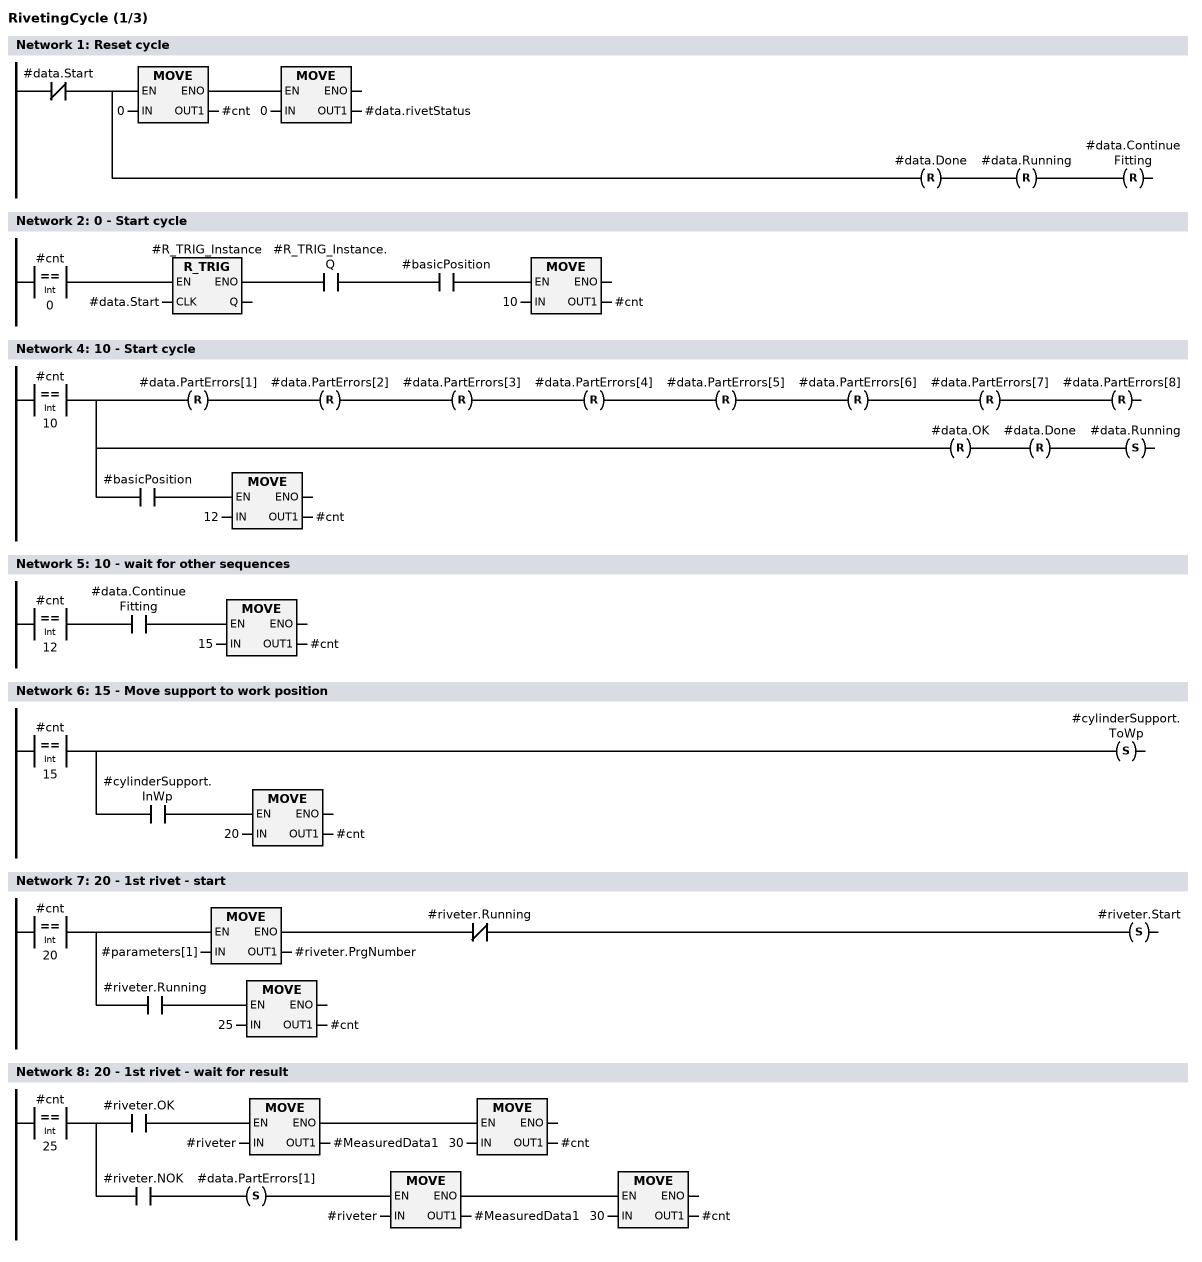
   RUNG wire#powerrail
      I_Contact( #data.Start )
      wire#w1
      Move(in := 0, out1 => #cnt)
      Move(in := 0, out1 => #data.rivetStatus)
   END_RUNG
   RUNG wire#w1
      R_Coil( #data.Done )
      R_Coil( #data.Running )
      R_Coil( #data.ContinueFitting )
   END_RUNG
   // the same network as SCL:
   IF NOT #data.Start THEN
       #cnt := 0;
       #data.rivetStatus := 0;
       #data.Done := FALSE;
       #data.Running := FALSE;
       #data.ContinueFitting := FALSE;
   END_IF;
END_REGION

REGION Network 2: 0 - Start cycle
   RUNG wire#powerrail
      { S7_Templates := "SrcType := Int" } EQ_Contact(in1 := #cnt, in2 := 0)
      #R_TRIG_Instance.R_TRIG(CLK := #data.Start, Q =>)
      Contact( #R_TRIG_Instance.Q )
      Contact( #basicPosition )
      Move(in := 10, out1 => #cnt)
   END_RUNG
   // the same network as SCL:
   #_w1 := #cnt = 0;
   #R_TRIG_Instance(EN := #_w1, CLK := #data.Start, ENO => #_w2);   // R_TRIG
   IF #_w2 AND #R_TRIG_Instance.Q AND #basicPosition THEN #cnt := 10; END_IF;
END_REGION

REGION Network 3 (SCL): 10 - Start cycle - init measured data
   IF #cnt = 10 THEN
       #MeasuredData1.Start := FALSE;
       #MeasuredData1.PrgNumber := 0;
       #MeasuredData1.Ready := FALSE;
       #MeasuredData1.Running := FALSE;
       #MeasuredData1.OK := FALSE;
       #MeasuredData1.NOK := FALSE;
       #MeasuredData1.H1OK := FALSE;
       #MeasuredData1.H2OK := FALSE;
       #MeasuredData1.TimeOK := FALSE;
       #MeasuredData1.StartError := FALSE;
       #MeasuredData1.LastH1 := 0.0;
       #MeasuredData1.LastH2 := 0.0;
       #MeasuredData1.LastTime := 0.0;
       #MeasuredData1.LastZ1 := 0.0;
       #MeasuredData1.Error := FALSE;
       #MeasuredData1.Z1OK := FALSE;
       #MeasuredData1.NewDataAfterStart := FALSE;
       #MeasuredData2 := #MeasuredData1;
   END_IF;
END_REGION

REGION Network 4: 10 - Start cycle
   RUNG wire#powerrail
      { S7_Templates := "SrcType := Int" } EQ_Contact(in1 := #cnt, in2 := 10)
      wire#w1
      R_Coil( #data.PartErrors[1] )
      R_Coil( #data.PartErrors[2] )
      R_Coil( #data.PartErrors[3] )
      R_Coil( #data.PartErrors[4] )
      R_Coil( #data.PartErrors[5] )
      R_Coil( #data.PartErrors[6] )
      R_Coil( #data.PartErrors[7] )
      R_Coil( #data.PartErrors[8] )
   END_RUNG
   RUNG wire#w1
      R_Coil( #data.OK )
      R_Coil( #data.Done )
      S_Coil( #data.Running )
   END_RUNG
   RUNG wire#w1
      Contact( #basicPosition )
      Move(in := 12, out1 => #cnt)
   END_RUNG
   // the same network as SCL:
   #_w1 := #cnt = 10;
   IF #_w1 THEN
       #data.PartErrors[1] := FALSE;
       #data.PartErrors[2] := FALSE;
       #data.PartErrors[3] := FALSE;
       #data.PartErrors[4] := FALSE;
       #data.PartErrors[5] := FALSE;
       #data.PartErrors[6] := FALSE;
       #data.PartErrors[7] := FALSE;
       #data.PartErrors[8] := FALSE;
       #data.OK := FALSE;
       #data.Done := FALSE;
       #data.Running := TRUE;
   END_IF;
   IF #_w1 AND #basicPosition THEN #cnt := 12; END_IF;
END_REGION

REGION Network 5: 10 - wait for other sequences
   RUNG wire#powerrail
      { S7_Templates := "SrcType := Int" } EQ_Contact(in1 := #cnt, in2 := 12)
      Contact( #data.ContinueFitting )
      Move(in := 15, out1 => #cnt)
   END_RUNG
   // the same network as SCL:
   IF (#cnt = 12) AND #data.ContinueFitting THEN #cnt := 15; END_IF;
END_REGION

REGION Network 6: 15 - Move support to work position
   RUNG wire#powerrail
      { S7_Templates := "SrcType := Int" } EQ_Contact(in1 := #cnt, in2 := 15)
      wire#w1
      S_Coil( #cylinderSupport.ToWp )
   END_RUNG
   RUNG wire#w1
      Contact( #cylinderSupport.InWp )
      Move(in := 20, out1 => #cnt)
   END_RUNG
   // the same network as SCL:
   #_w1 := #cnt = 15;
   IF #_w1 THEN #cylinderSupport.ToWp := TRUE; END_IF;
   IF #_w1 AND #cylinderSupport.InWp THEN #cnt := 20; END_IF;
END_REGION

REGION Network 7: 20 - 1st rivet - start
   RUNG wire#powerrail
      { S7_Templates := "SrcType := Int" } EQ_Contact(in1 := #cnt, in2 := 20)
      wire#w1
      Move(in := #parameters[1], out1 => #riveter.PrgNumber)
      I_Contact( #riveter.Running )
      S_Coil( #riveter.Start )
   END_RUNG
   RUNG wire#w1
      Contact( #riveter.Running )
      Move(in := 25, out1 => #cnt)
   END_RUNG
   // the same network as SCL:
   #_w1 := #cnt = 20;
   IF #_w1 THEN #riveter.PrgNumber := #parameters[1]; END_IF;
   IF #_w1 AND NOT #riveter.Running THEN #riveter.Start := TRUE; END_IF;
   IF #_w1 AND #riveter.Running THEN #cnt := 25; END_IF;
END_REGION

REGION Network 8: 20 - 1st rivet - wait for result
   RUNG wire#powerrail
      { S7_Templates := "SrcType := Int" } EQ_Contact(in1 := #cnt, in2 := 25)
      wire#w1
      Contact( #riveter.OK )
      Move(in := #riveter, out1 => #MeasuredData1)
      Move(in := 30, out1 => #cnt)
   END_RUNG
   RUNG wire#w1
      Contact( #riveter.NOK )
      S_Coil( #data.PartErrors[1] )
      Move(in := #riveter, out1 => #MeasuredData1)
      Move(in := 30, out1 => #cnt)
   END_RUNG
   // the same network as SCL:
   #_w1 := #cnt = 25;
   IF #_w1 AND #riveter.OK THEN
       #MeasuredData1 := #riveter;
       #cnt := 30;
   END_IF;
   IF #_w1 AND #riveter.NOK THEN
       #data.PartErrors[1] := TRUE;
       #MeasuredData1 := #riveter;
       #cnt := 30;
   END_IF;
END_REGION

REGION Network 9: 30 - Move support to base position
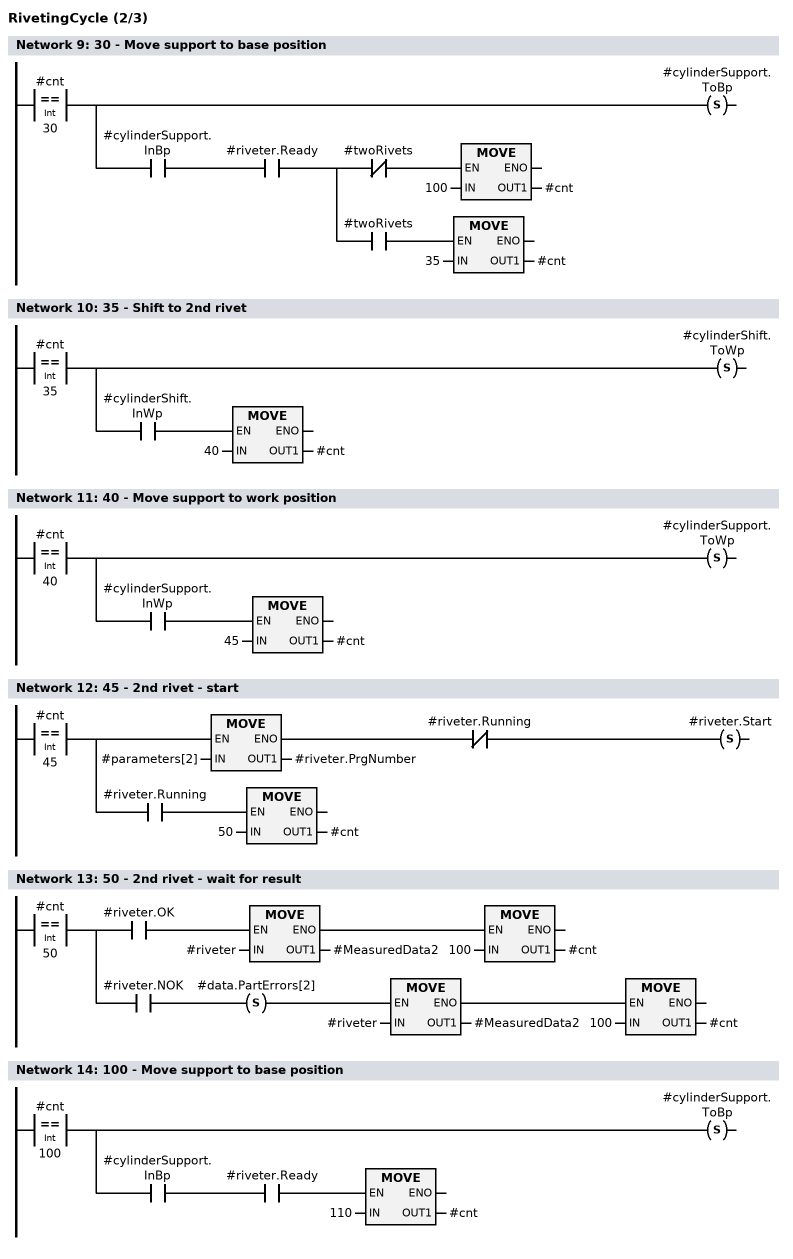
   RUNG wire#powerrail
      { S7_Templates := "SrcType := Int" } EQ_Contact(in1 := #cnt, in2 := 30)
      wire#w1
      S_Coil( #cylinderSupport.ToBp )
   END_RUNG
   RUNG wire#w1
      Contact( #cylinderSupport.InBp )
      Contact( #riveter.Ready )
      wire#w2
      I_Contact( #twoRivets )
      Move(in := 100, out1 => #cnt)
   END_RUNG
   RUNG wire#w2
      Contact( #twoRivets )
      Move(in := 35, out1 => #cnt)
   END_RUNG
   // the same network as SCL:
   #_w1 := #cnt = 30;
   IF #_w1 THEN #cylinderSupport.ToBp := TRUE; END_IF;
   #_w2 := #_w1 AND #cylinderSupport.InBp AND #riveter.Ready;
   IF #_w2 AND NOT #twoRivets THEN #cnt := 100; END_IF;
   IF #_w2 AND #twoRivets THEN #cnt := 35; END_IF;
END_REGION

REGION Network 10: 35 - Shift to 2nd rivet
   RUNG wire#powerrail
      { S7_Templates := "SrcType := Int" } EQ_Contact(in1 := #cnt, in2 := 35)
      wire#w1
      S_Coil( #cylinderShift.ToWp )
   END_RUNG
   RUNG wire#w1
      Contact( #cylinderShift.InWp )
      Move(in := 40, out1 => #cnt)
   END_RUNG
   // the same network as SCL:
   #_w1 := #cnt = 35;
   IF #_w1 THEN #cylinderShift.ToWp := TRUE; END_IF;
   IF #_w1 AND #cylinderShift.InWp THEN #cnt := 40; END_IF;
END_REGION

REGION Network 11: 40 - Move support to work position
   RUNG wire#powerrail
      { S7_Templates := "SrcType := Int" } EQ_Contact(in1 := #cnt, in2 := 40)
      wire#w1
      S_Coil( #cylinderSupport.ToWp )
   END_RUNG
   RUNG wire#w1
      Contact( #cylinderSupport.InWp )
      Move(in := 45, out1 => #cnt)
   END_RUNG
   // the same network as SCL:
   #_w1 := #cnt = 40;
   IF #_w1 THEN #cylinderSupport.ToWp := TRUE; END_IF;
   IF #_w1 AND #cylinderSupport.InWp THEN #cnt := 45; END_IF;
END_REGION

REGION Network 12: 45 - 2nd rivet - start
   RUNG wire#powerrail
      { S7_Templates := "SrcType := Int" } EQ_Contact(in1 := #cnt, in2 := 45)
      wire#w1
      Move(in := #parameters[2], out1 => #riveter.PrgNumber)
      I_Contact( #riveter.Running )
      S_Coil( #riveter.Start )
   END_RUNG
   RUNG wire#w1
      Contact( #riveter.Running )
      Move(in := 50, out1 => #cnt)
   END_RUNG
   // the same network as SCL:
   #_w1 := #cnt = 45;
   IF #_w1 THEN #riveter.PrgNumber := #parameters[2]; END_IF;
   IF #_w1 AND NOT #riveter.Running THEN #riveter.Start := TRUE; END_IF;
   IF #_w1 AND #riveter.Running THEN #cnt := 50; END_IF;
END_REGION

REGION Network 13: 50 - 2nd rivet - wait for result
   RUNG wire#powerrail
      { S7_Templates := "SrcType := Int" } EQ_Contact(in1 := #cnt, in2 := 50)
      wire#w1
      Contact( #riveter.OK )
      Move(in := #riveter, out1 => #MeasuredData2)
      Move(in := 100, out1 => #cnt)
   END_RUNG
   RUNG wire#w1
      Contact( #riveter.NOK )
      S_Coil( #data.PartErrors[2] )
      Move(in := #riveter, out1 => #MeasuredData2)
      Move(in := 100, out1 => #cnt)
   END_RUNG
   // the same network as SCL:
   #_w1 := #cnt = 50;
   IF #_w1 AND #riveter.OK THEN
       #MeasuredData2 := #riveter;
       #cnt := 100;
   END_IF;
   IF #_w1 AND #riveter.NOK THEN
       #data.PartErrors[2] := TRUE;
       #MeasuredData2 := #riveter;
       #cnt := 100;
   END_IF;
END_REGION

REGION Network 14: 100 - Move support to base position
   RUNG wire#powerrail
      { S7_Templates := "SrcType := Int" } EQ_Contact(in1 := #cnt, in2 := 100)
      wire#w1
      S_Coil( #cylinderSupport.ToBp )
   END_RUNG
   RUNG wire#w1
      Contact( #cylinderSupport.InBp )
      Contact( #riveter.Ready )
      Move(in := 110, out1 => #cnt)
   END_RUNG
   // the same network as SCL:
   #_w1 := #cnt = 100;
   IF #_w1 THEN #cylinderSupport.ToBp := TRUE; END_IF;
   IF #_w1 AND #cylinderSupport.InBp AND #riveter.Ready THEN #cnt := 110; END_IF;
END_REGION

REGION Network 15: 110 - Shift to base position
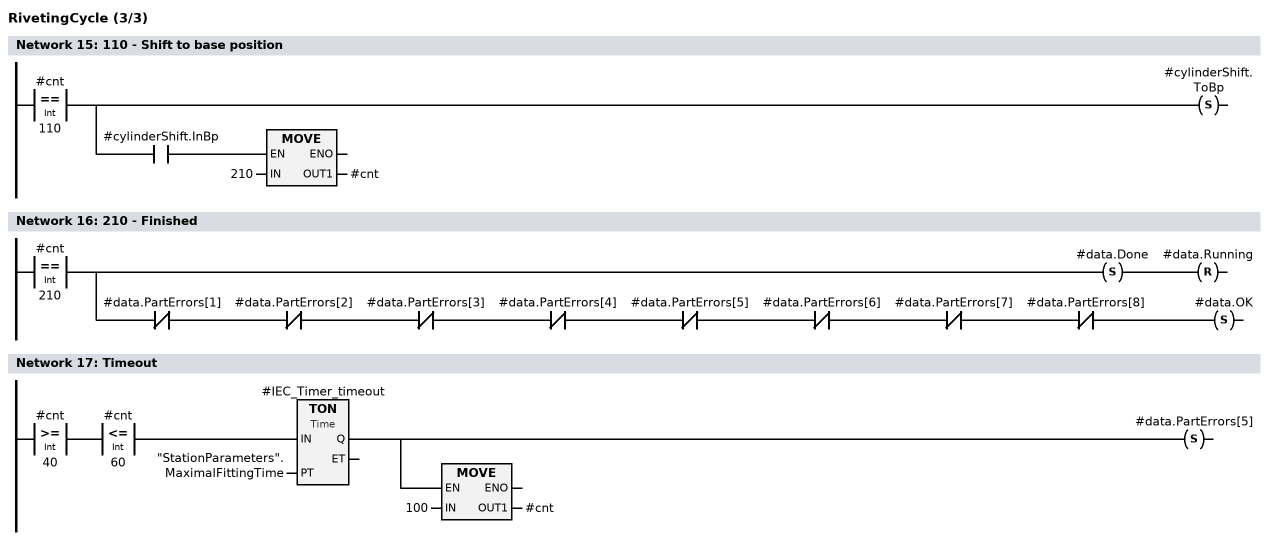
   RUNG wire#powerrail
      { S7_Templates := "SrcType := Int" } EQ_Contact(in1 := #cnt, in2 := 110)
      wire#w1
      S_Coil( #cylinderShift.ToBp )
   END_RUNG
   RUNG wire#w1
      Contact( #cylinderShift.InBp )
      Move(in := 210, out1 => #cnt)
   END_RUNG
   // the same network as SCL:
   #_w1 := #cnt = 110;
   IF #_w1 THEN #cylinderShift.ToBp := TRUE; END_IF;
   IF #_w1 AND #cylinderShift.InBp THEN #cnt := 210; END_IF;
END_REGION

REGION Network 16: 210 - Finished
   RUNG wire#powerrail
      { S7_Templates := "SrcType := Int" } EQ_Contact(in1 := #cnt, in2 := 210)
      wire#w1
      S_Coil( #data.Done )
      R_Coil( #data.Running )
   END_RUNG
   RUNG wire#w1
      I_Contact( #data.PartErrors[1] )
      I_Contact( #data.PartErrors[2] )
      I_Contact( #data.PartErrors[3] )
      I_Contact( #data.PartErrors[4] )
      I_Contact( #data.PartErrors[5] )
      I_Contact( #data.PartErrors[6] )
      I_Contact( #data.PartErrors[7] )
      I_Contact( #data.PartErrors[8] )
      S_Coil( #data.OK )
   END_RUNG
   // the same network as SCL:
   #_w1 := #cnt = 210;
   IF #_w1 THEN
       #data.Done := TRUE;
       #data.Running := FALSE;
   END_IF;
   IF #_w1 AND NOT #data.PartErrors[1] AND NOT #data.PartErrors[2] AND NOT #data.PartErrors[3] AND NOT #data.PartErrors[4] AND NOT #data.PartErrors[5] AND NOT #data.PartErrors[6] AND NOT #data.PartErrors[7] AND NOT #data.PartErrors[8] THEN
       #data.OK := TRUE;
   END_IF;
END_REGION

REGION Network 17: Timeout
   RUNG wire#powerrail
      { S7_Templates := "SrcType := Int" } GE_Contact(in1 := #cnt, in2 := 40)
      { S7_Templates := "SrcType := Int" } LE_Contact(in1 := #cnt, in2 := 60)
      { S7_Templates := "time_type := Time" } #IEC_Timer_timeout.TON(pt := "StationParameters".MaximalFittingTime, et =>)
      wire#w1
      S_Coil( #data.PartErrors[5] )
   END_RUNG
   RUNG wire#w1
      Move(in := 100, out1 => #cnt)
   END_RUNG
   // the same network as SCL:
   #IEC_Timer_timeout(IN := (#cnt >= 40) AND (#cnt <= 60), PT := "StationParameters".MaximalFittingTime);   // TON
   IF #IEC_Timer_timeout.Q THEN
       #data.PartErrors[5] := TRUE;
       #cnt := 100;
   END_IF;
END_REGION
END_FUNCTION_BLOCK

FUNCTION_BLOCK "Manipulator_main"
{ S7_Optimized_Access := 'TRUE' }
VERSION : 0.1
   VAR 
      PUT_Instance {InstructionName := 'PUT'; LibVersion := '1.3'; S7_SetPoint := 'False'} : PUT;
      GET_Instance {InstructionName := 'GET'; LibVersion := '1.3'; S7_SetPoint := 'False'} : GET;
      GetStatusMem : Word;
      PutStatusMem : Word;
      GetCounterNDR : ULInt;
      PutCounterDone : ULInt;
      GetCounterNDR_last : ULInt;
      PutCounterDone_last : ULInt;
      GetCommOK : Bool;
      PutCommOK : Bool;
      R_TRIG_GetNDR {InstructionName := 'R_TRIG'; LibVersion := '1.0'; S7_SetPoint := 'False'} : R_TRIG;
      R_TRIG_PutDone {InstructionName := 'R_TRIG'; LibVersion := '1.0'; S7_SetPoint := 'False'} : R_TRIG;
      IEC_Timer_GetCommOK {InstructionName := 'TOF_TIME'; LibVersion := '1.0'} : TOF_TIME;
      IEC_Timer_PutCommOK {InstructionName := 'TOF_TIME'; LibVersion := '1.0'} : TOF_TIME;
   END_VAR


BEGIN
	REGION GET
	    #GET_Instance(ID := W#16#100,
	                  ADDR_1 := P#db1002.dbx0.0 byte 100,
	                  RD_1 := P#db1002.dbx0.0 byte 100);
	    IF #GET_Instance.ERROR THEN
	        #GetStatusMem := #GET_Instance.STATUS;
	    END_IF;
	    IF #GET_Instance.NDR THEN
	        #GetStatusMem := 0;
	    END_IF;
	    #R_TRIG_GetNDR(CLK := #GET_Instance.NDR);
	    IF #R_TRIG_GetNDR.Q THEN
	        #GetCounterNDR := #GetCounterNDR + 1;
	    END_IF;
	    #GET_Instance.REQ := NOT #GET_Instance.REQ;
	END_REGION
	
	"Manipulator<<<Main".counter := "Manipulator>>>Main".counter + 1;
	"Manipulator<<<Main".robotOutOfZone := "iR1OutOfSt4" ;
	"Manipulator<<<Main".airSupplyStatus := "safety_signals".doorUnlocked;
	
	IF "DB_MainData".MachineMode >= 3 THEN
	    "Manipulator<<<Main".automaticModeActive := TRUE;
	END_IF;
	    
	
	REGION comm diagnostic
	    #IEC_Timer_GetCommOK(IN := #GetCounterNDR <> #GetCounterNDR_last,
	   PT := t#1s,
	   Q => #GetCommOK);
	    #IEC_Timer_PutCommOK(IN := #PutCounterDone <> #PutCounterDone_last,
	   PT := t#1s,
	   Q => #PutCommOK);
	    #GetCounterNDR_last := #GetCounterNDR;
	    #PutCounterDone_last := #PutCounterDone;
	END_REGION
	
	REGION PUT
	    #PUT_Instance(ID := W#16#100,
	                  ADDR_1 := P#db1001.dbx0.0 byte 100,
	                  SD_1 := P#db1001.dbx0.0 byte 100);
	    #PUT_Instance.REQ := NOT #PUT_Instance.REQ;
	    IF #PUT_Instance.ERROR THEN
	        #PutStatusMem := #PUT_Instance.STATUS;
	    END_IF;
	    IF #PUT_Instance.DONE THEN
	        #PutStatusMem := 0;
	    END_IF;
	    #R_TRIG_PutDone(CLK:=#PUT_Instance.DONE);
	    IF #R_TRIG_PutDone.Q THEN
	        #PutCounterDone := #PutCounterDone + 1;
	    END_IF;
	END_REGION
	
	
	
	
END_FUNCTION_BLOCK

FUNCTION_BLOCK "SlidesMain"   // FB25, LAD
{ S7_Optimized_Access := 'TRUE' }
VERSION : 0.1
// stored: AutoNumber true, IsIECCheckEnabled false, IsRetainMemResEnabled false, MemoryReserve 100, SetENOAutomatically false, UDAEnableTagReadback false
   VAR
      R_TRIG_Instance { S7_SetPoint := 'True'} : R_TRIG;
      IEC_Timer_0_Instance { S7_SetPoint := 'True'} : TON_TIME;
      IEC_Timer_0_Instance_1 { S7_SetPoint := 'True'} : TOF_TIME;
      IEC_Timer_0_Instance_3 { S7_SetPoint := 'True'} : TON_TIME;
      IEC_Timer_0_Instance_5 { S7_SetPoint := 'True'} : TON_TIME;
   END_VAR
BEGIN

REGION Network 1 (SCL): NOK box from part holders
   //Check amount of parts in stock
   IF "PartHolderData".NOKBoxAmount >= "StationParameters".NOKBoxSize THEN
       "PartHolderData".NOKBoxFull := true;
   ELSE
       "PartHolderData".NOKBoxFull := FALSE;
   END_IF;

   //NOK Box signal with delay
   #R_TRIG_Instance(CLK:=NOT "iNokPartOpticalSensor");
   IF #R_TRIG_Instance.Q THEN
       "PartHolderData".NOKBoxActivated := true;
   END_IF;
   #IEC_Timer_0_Instance(IN:="PartHolderData".NOKBoxActivated,
                         PT:=t#2s);
   IF #IEC_Timer_0_Instance.Q THEN
       "PartHolderData".NOKBoxActivated := false;
   END_IF;

   //Box presence with delay
   #IEC_Timer_0_Instance_1(IN:="iNokBoxPresent",
                           PT:=t#1s,
                           Q=>"PartHolderData".NOKBoxPesent);

   //Error NOK box signal sensor
   #IEC_Timer_0_Instance_3(IN:=NOT "iNokPartOpticalSensor",
                           PT:=t#3s);
   IF #IEC_Timer_0_Instance_3.Q AND "PartHolderData".NOKBoxPesent THEN
       "SetAlarm"(AlarmNumber := 42,
                  Cell := 1,
                  Station := 99);
       ;
   END_IF;

   #IEC_Timer_0_Instance_5(IN:=NOT "iNokBoxPresent",
                           PT:=t#3s);
   IF #IEC_Timer_0_Instance_5.Q THEN
       "SetAlarm"(AlarmNumber := 40,
                  Cell := 1,
                  Station := 99);
       ;
   END_IF;

   IF "PartHolderData".NOKBoxFull THEN
       "SetAlarm"(AlarmNumber := 43,
                  Cell := 1,
                  Station := 99);
   END_IF;

   //Reset holders amounts
   "PartHolderData".ConfirmEmptyNOKBox := "PartHolderData".NOKBoxFull;
   IF "PartHolderData".EmptyNOKBoxConfirmed THEN
       "PartHolderData".NOKBoxAmount := 0;
   END_IF;
   "PartHolderData".EmptyNOKBoxConfirmed := false;
END_REGION
END_FUNCTION_BLOCK

FUNCTION_BLOCK "HMIMain"
{ S7_Optimized_Access := 'TRUE' }
VERSION : 0.1
   VAR 
      res : Bool;
   END_VAR


BEGIN
	//screen number
	"HMIData".HMI.ActualScreenNumber:="HMIData".HMI.ScreenData[2];
	
	//Manual command
	"HMIData".ManualCommand := 0;
	//"ModeSelectionData".ManualMode := true;
	
	IF "HMIData".ManualCommandHMI > 0 AND "SystemHMI".ManualMode THEN
	    "HMIData".ManualCommand := "HMIData".ManualCommandHMI;
	    "HMIData".ManualCommandHMI := 0;
	ELSE
	    "HMIData".ManualCommandHMI := 0;
	END_IF;
	
END_FUNCTION_BLOCK

FUNCTION_BLOCK "ModeSelection"   // FB38, GRAPH
VERSION : 0.1
// stored: AcknowledgeErrorsRequired true, AutoNumber true, GraphVersion 6.0, InitialValuesAcquisition false, IsIECCheckEnabled false, LanguageInNetworks LAD, LockOperatingMode false, PermanentILProcessingInMANMode false, SetENOAutomatically false, SkipSteps false, UDAEnableTagReadback false, WithAlarmHandling true
   // inherited from GRAPH_BASE
   VAR
      OFF_SQ_BASE : Bool;
   END_VAR
   VAR_INPUT
      iSafetyOKauto : Bool;
      iSafetyOKmanual : Bool;
      iBasePosition : Bool;
      iPozadavekZastavitOdDveri : Bool;
      iLinkaZastavena : Bool;
      iLinkaPrazdna : Bool;
      iBaseInManualMode : Bool;
      OFF_SQ { ExternalAccessible := 'False'; ExternalVisible := 'False'; ExternalWritable := 'False'} : Bool := false;   // Turn sequence off
      INIT_SQ { ExternalAccessible := 'False'; ExternalVisible := 'False'; ExternalWritable := 'False'} : Bool := false;   // Set sequence to initial state
      ACK_EF { ExternalAccessible := 'False'; ExternalVisible := 'False'; ExternalWritable := 'False'} : Bool := false;   // Acknowledge all errors and faults
      S_PREV { ExternalAccessible := 'False'; ExternalVisible := 'False'; ExternalWritable := 'False'} : Bool := false;   // Output previous step in parameter S_NO
      S_NEXT { ExternalAccessible := 'False'; ExternalVisible := 'False'; ExternalWritable := 'False'} : Bool := false;   // Indicate next step in parameter S_NO
      SW_AUTO { ExternalAccessible := 'False'; ExternalVisible := 'False'; ExternalWritable := 'False'} : Bool := false;   // Automatic mode
      SW_TAP { ExternalAccessible := 'False'; ExternalVisible := 'False'; ExternalWritable := 'False'} : Bool := false;   // Semiautomatic/switch with transition
      SW_TOP { ExternalAccessible := 'False'; ExternalVisible := 'False'; ExternalWritable := 'False'} : Bool := false;   // Semiautomatic/ignore transition
      SW_MAN { ExternalAccessible := 'False'; ExternalVisible := 'False'; ExternalWritable := 'False'} : Bool := false;   // Manual mode
      S_SEL { ExternalAccessible := 'False'; ExternalVisible := 'False'; ExternalWritable := 'False'} : Int := 0;   // Select step to be output to S_NO
      S_ON { ExternalAccessible := 'False'; ExternalVisible := 'False'; ExternalWritable := 'False'} : Bool := false;   // Activate step indicated in S_NO
      S_OFF { ExternalAccessible := 'False'; ExternalVisible := 'False'; ExternalWritable := 'False'} : Bool := false;   // Deactivate step indicated S_NO
      T_PUSH { ExternalAccessible := 'False'; ExternalVisible := 'False'; ExternalWritable := 'False'} : Bool := false;   // Enable transition to switch in semi automatic mode
   END_VAR
   VAR_OUTPUT
      S_NO { ExternalAccessible := 'False'; ExternalVisible := 'False'; ExternalWritable := 'False'} : Int := 0;   // Step number
      S_MORE { ExternalAccessible := 'False'; ExternalVisible := 'False'; ExternalWritable := 'False'} : Bool := false;   // More steps are available and can be shown in S_NO
      S_ACTIVE { ExternalAccessible := 'False'; ExternalVisible := 'False'; ExternalWritable := 'False'} : Bool := false;   // Step indicated in S_NO is active
      ERR_FLT { ExternalAccessible := 'False'; ExternalVisible := 'False'; ExternalWritable := 'False'} : Bool := false;   // Interlock or supervision group error
      AUTO_ON { ExternalAccessible := 'False'; ExternalVisible := 'False'; ExternalWritable := 'False'} : Bool := false;   // Automatic mode is active
      TAP_ON { ExternalAccessible := 'False'; ExternalVisible := 'False'; ExternalWritable := 'False'} : Bool := false;   // Semiautomatic mode/step with transition enabled
      TOP_ON { ExternalAccessible := 'False'; ExternalVisible := 'False'; ExternalWritable := 'False'} : Bool := false;   // Semiautomatic mode/ignore transition enabled
      MAN_ON { ExternalAccessible := 'False'; ExternalVisible := 'False'; ExternalWritable := 'False'} : Bool := false;   // Manual mode is active
   END_VAR
   VAR
      dummy : Bool;
   END_VAR
   VAR RETAIN
      mode : "udtModes";
   END_VAR
   VAR
      PrevMode : Int;
      F_TRIG_semiauto_switch { S7_SetPoint := 'True'} : F_TRIG;
      F_TRIG_switchAuto { S7_SetPoint := 'True'} : F_TRIG;
   END_VAR
BEGIN
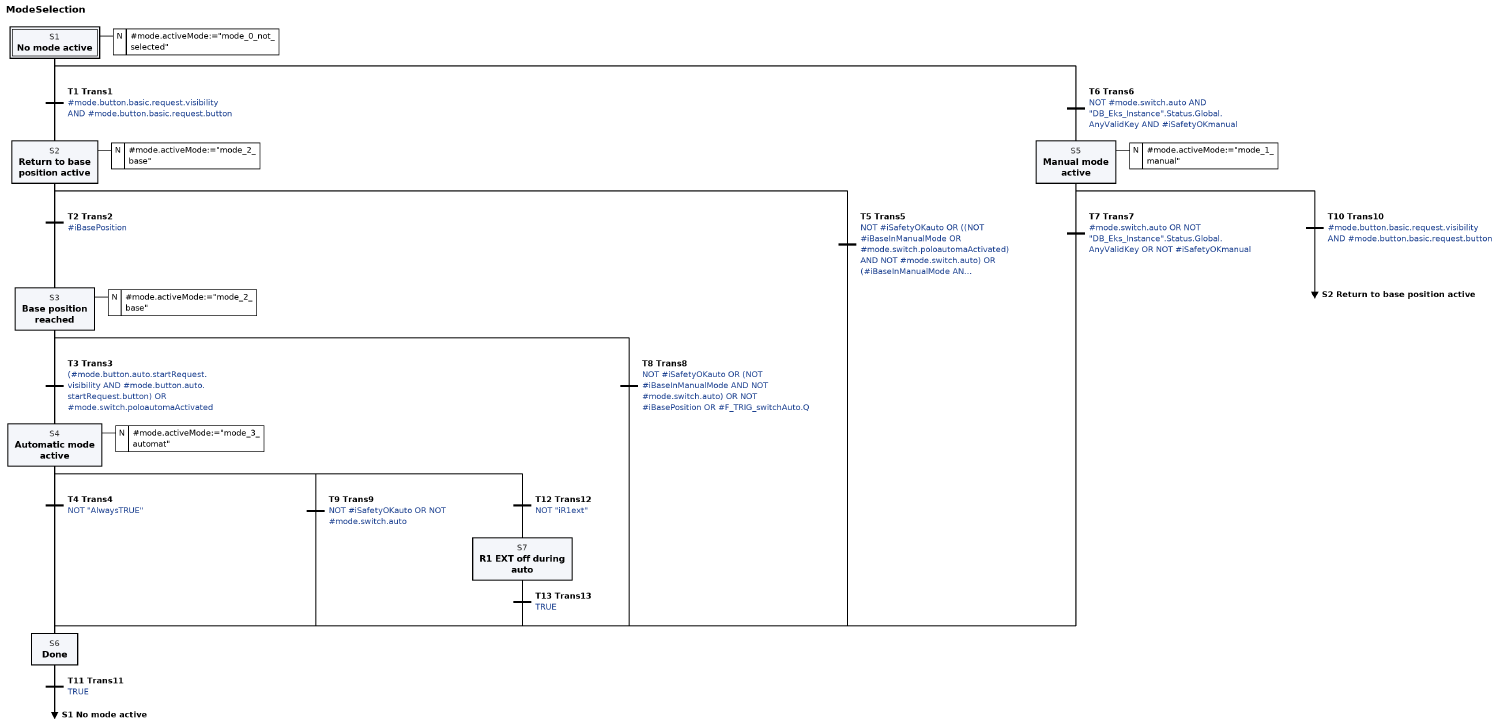
   // permanent pre-instructions
   NETWORK 1
   TITLE = mode init
      "ModeSelection_DB".mode.activeMode := "mode_0_not_selected";
   NETWORK 2
   TITLE = button visibility
      #mode.button.basic.request.visibility := #iSafetyOKauto AND ((#mode.switch.auto AND #"No mode active".X AND (NOT #iBaseInManualMode OR #mode.switch.poloautomaActivated)) OR (NOT #mode.switch.auto AND #"Manual mode active".X AND #iBaseInManualMode AND NOT #mode.switch.poloautomaActivated));
      #mode.button.auto.startRequest.visibility := #iSafetyOKauto AND #mode.switch.auto AND #"Base position reached".X AND NOT "SystemHMI".AlarmActive;
   NETWORK 3
   TITLE = semiauto switch off detection
      #F_TRIG_semiauto_switch(CLK := #mode.switch.poloautomaActivated);   // F_TRIG
   NETWORK 4
      #F_TRIG_switchAuto(CLK := #mode.switch.auto);   // F_TRIG

   // sequencer 1
   INITIAL_STEP "No mode active":   // S1, max time T#10S, warning time T#7S
              N    #mode.activeMode:="mode_0_not_selected"
   END_STEP
   TRANSITION Trans1 FROM "No mode active" TO "Return to base position active"   // T1
      := #mode.button.basic.request.visibility AND #mode.button.basic.request.button;
   END_TRANSITION
   TRANSITION Trans6 FROM "No mode active" TO "Manual mode active"   // T6
      := NOT #mode.switch.auto AND "DB_Eks_Instance".Status.Global.AnyValidKey AND #iSafetyOKmanual;
   END_TRANSITION
   STEP "Return to base position active":   // S2, max time T#10S, warning time T#7S
              N    #mode.activeMode:="mode_2_base"
   END_STEP
   TRANSITION Trans2 FROM "Return to base position active" TO "Base position reached"   // T2
      := #iBasePosition;
   END_TRANSITION
   TRANSITION Trans5 FROM "Return to base position active" TO Done   // T5
      := NOT #iSafetyOKauto OR ((NOT #iBaseInManualMode OR #mode.switch.poloautomaActivated) AND NOT #mode.switch.auto) OR (#iBaseInManualMode AND #mode.switch.auto AND NOT #mode.switch.poloautomaActivated) OR #F_TRIG_semiauto_switch.Q;
   END_TRANSITION
   STEP "Base position reached":   // S3, max time T#10S, warning time T#7S
              N    #mode.activeMode:="mode_2_base"
   END_STEP
   TRANSITION Trans3 FROM "Base position reached" TO "Automatic mode active"   // T3
      := (#mode.button.auto.startRequest.visibility AND #mode.button.auto.startRequest.button) OR #mode.switch.poloautomaActivated;
   END_TRANSITION
   TRANSITION Trans8 FROM "Base position reached" TO Done   // T8
      := NOT #iSafetyOKauto OR (NOT #iBaseInManualMode AND NOT #mode.switch.auto) OR NOT #iBasePosition OR #F_TRIG_switchAuto.Q;
   END_TRANSITION
   STEP "Automatic mode active":   // S4, max time T#10S, warning time T#7S
              N    #mode.activeMode:="mode_3_automat"
   END_STEP
   TRANSITION Trans4 FROM "Automatic mode active" TO Done   // T4
      := NOT "AlwaysTRUE";
   END_TRANSITION
   TRANSITION Trans9 FROM "Automatic mode active" TO Done   // T9
      := NOT #iSafetyOKauto OR NOT #mode.switch.auto;
   END_TRANSITION
   TRANSITION Trans12 FROM "Automatic mode active" TO "R1 EXT off during auto"   // T12
      := NOT "iR1ext";
   END_TRANSITION
   STEP "Manual mode active":   // S5, max time T#10S, warning time T#7S
              N    #mode.activeMode:="mode_1_manual"
   END_STEP
   TRANSITION Trans7 FROM "Manual mode active" TO Done   // T7
      := #mode.switch.auto OR NOT "DB_Eks_Instance".Status.Global.AnyValidKey OR NOT #iSafetyOKmanual;
   END_TRANSITION
   TRANSITION Trans10 FROM "Manual mode active" TO "Return to base position active"   // T10, jump
      := #mode.button.basic.request.visibility AND #mode.button.basic.request.button;
   END_TRANSITION
   STEP Done:   // S6, max time T#10S, warning time T#7S
   END_STEP
   TRANSITION Trans11 FROM Done TO "No mode active"   // T11, jump
      := TRUE;
   END_TRANSITION
   STEP "R1 EXT off during auto":   // S7, max time T#10S, warning time T#7S
   END_STEP
   TRANSITION Trans13 FROM "R1 EXT off during auto" TO Done   // T13
      := TRUE;
   END_TRANSITION

   // permanent post-instructions
   NETWORK 1
   TITLE = semiauto mode
      IF ((#mode.activeMode = "mode_2_base") OR (#mode.activeMode = "mode_3_automat")) AND #mode.switch.poloautomaActivated THEN
          #mode.activeMode := "mode_4_semiautomat";
      END_IF;
   NETWORK 2
   TITLE = previous mode
      #mode.modeChanged := #mode.activeMode <> #PrevMode;
      #PrevMode := #mode.activeMode;
END_FUNCTION_BLOCK

FUNCTION_BLOCK "sequences_main"
{ S7_Optimized_Access := 'TRUE' }
VERSION : 0.1

BEGIN
	
	"sq_robot_"(OFF_SQ := NOT "sq_robot_".INIT_SQ,
	            INIT_SQ := "ModeSelection_DB".mode.activeMode = "mode_2_base" OR
	            "ModeSelection_DB".mode.activeMode = "mode_3_automat" OR
	            "ModeSelection_DB".mode.activeMode = "mode_4_semiautomat",
	            ACK_EF := "Alarms".Reset);
	
	"sq_carousel_main_"(OFF_SQ := NOT "sq_carousel_main_".INIT_SQ,
	                    INIT_SQ := "ModeSelection_DB".mode.activeMode = "mode_2_base" OR
	                    "ModeSelection_DB".mode.activeMode = "mode_3_automat" OR
	                    "ModeSelection_DB".mode.activeMode = "mode_4_semiautomat",
	                    ACK_EF := "Alarms".Reset);
	
	"sq_carousel_insertion_st1"(OFF_SQ := NOT "sq_carousel_insertion_st1".INIT_SQ,
	                            INIT_SQ := "ModeSelection_DB".mode.activeMode = "mode_2_base" OR
	                            "ModeSelection_DB".mode.activeMode = "mode_3_automat" OR
	                            "ModeSelection_DB".mode.activeMode = "mode_4_semiautomat",
	                            ACK_EF := "Alarms".Reset);
	
	"sq_carousel_unloading_st2"(OFF_SQ := NOT "sq_carousel_unloading_st2".INIT_SQ,
	                            INIT_SQ := "ModeSelection_DB".mode.activeMode = "mode_2_base" OR
	                            "ModeSelection_DB".mode.activeMode = "mode_3_automat" OR
	                            "ModeSelection_DB".mode.activeMode = "mode_4_semiautomat",
	                            ACK_EF := "Alarms".Reset);
	
	"sq_fitting_station_st3"(OFF_SQ := NOT "sq_fitting_station_st3".INIT_SQ,
	                         INIT_SQ := "ModeSelection_DB".mode.activeMode = "mode_2_base" OR
	                         "ModeSelection_DB".mode.activeMode = "mode_3_automat" OR
	                         "ModeSelection_DB".mode.activeMode = "mode_4_semiautomat",
	                         ACK_EF := "Alarms".Reset);
	
	"sq_autoeject_DB"(OFF_SQ := NOT "sq_autoeject_DB".INIT_SQ,
	                  INIT_SQ := "ModeSelection_DB".mode.activeMode = "mode_2_base" OR
	                  "ModeSelection_DB".mode.activeMode = "mode_3_automat" OR
	                  "ModeSelection_DB".mode.activeMode = "mode_4_semiautomat",
	                  ACK_EF := "Alarms".Reset);
	
	"sq_hanger_manipulator"(OFF_SQ := NOT "sq_hanger_manipulator".INIT_SQ,
	                    INIT_SQ := "ModeSelection_DB".mode.activeMode = "mode_2_base" OR
	                    "ModeSelection_DB".mode.activeMode = "mode_3_automat" OR
	                    "ModeSelection_DB".mode.activeMode = "mode_4_semiautomat",
	                    ACK_EF := "Alarms".Reset);
	
	
	
	"PartsDataTransfer_DB"();
	
	
	
	"sq_autoeject_DB".base :=
	"DevicesData"."TA1-3MA".AxisRef AND
	"DevicesData"."TA1-3MA".data.zones.inNOKpos AND
	"DevicesData".Cylinders["MM104_AutoejectGripperLifting"].InBp AND
	(
	NOT "AutoPositions".AE_Gripper.PartPresent AND
	NOT "iAEtubePresentFront" AND NOT "iAEtubePresentRear" AND
	"DevicesData".Cylinders["MM2500_GrippingTubeFront"].InBp AND
	"DevicesData".Cylinders["MM2520_HoldingSidememberInsideLeft"].InBp AND
	"DevicesData".Cylinders["MM2540_HoldingSidememberOutsideLeft"].InBp
	OR
	"AutoPositions".AE_Gripper.PartPresent AND
	"iAEtubePresentFront" AND "iAEtubePresentRear" AND
	"DevicesData".Cylinders["MM2500_GrippingTubeFront"].InWp AND
	"DevicesData".Cylinders["MM2520_HoldingSidememberInsideLeft"].InWp AND
	"DevicesData".Cylinders["MM2540_HoldingSidememberOutsideLeft"].InWp
	);
	
	
	IF NOT "SystemHMI".AutomaticMode THEN
	    "AutoInfo".EndProduction := FALSE;
	END_IF;
	
	
	
	
	
	
	
	
	
	
	
	
	
	
	
	
	
	
	
	
	
	
END_FUNCTION_BLOCK

FUNCTION_BLOCK "ParametersLimits"
{ S7_Optimized_Access := 'TRUE' }
VERSION : 0.1
   VAR RETAIN
      limits { S7_SetPoint := 'False'} : "udt_parametersLimits";
   END_VAR

   VAR_TEMP 
      i : Int;
   END_VAR


BEGIN
	#limits.ServoPositions[0].min := 5000;
	#limits.ServoPositions[0].max := 15000;
	#limits.ServoPositions[1].min := 780000;
	#limits.ServoPositions[1].max := 790000;
	#limits.ServoPositions[2].min := 1508000;
	#limits.ServoPositions[2].max := 1518000;
	
	FOR #i := 0 TO 9 DO
	    "StationParameters".ServoPositions[#i] :=
	    LIMIT(MN := #limits.ServoPositions[#i].min, IN := "StationParameters".ServoPositions[#i], MX := #limits.ServoPositions[#i].max);
	END_FOR;
	
	
END_FUNCTION_BLOCK

FUNCTION_BLOCK "Lamps"   // FB7, LAD
{ S7_Optimized_Access := 'TRUE' }
VERSION : 0.1
// stored: AutoNumber true, IsIECCheckEnabled false, IsRetainMemResEnabled false, MemoryReserve 100, SetENOAutomatically false, UDAEnableTagReadback false
   VAR
      R_TRIG_Instance { S7_SetPoint := 'True'} : R_TRIG;
      IEC_Timer_0_Instance { S7_SetPoint := 'True'} : TON_TIME;
   END_VAR
BEGIN

REGION Network 1: Lighthouse lamps
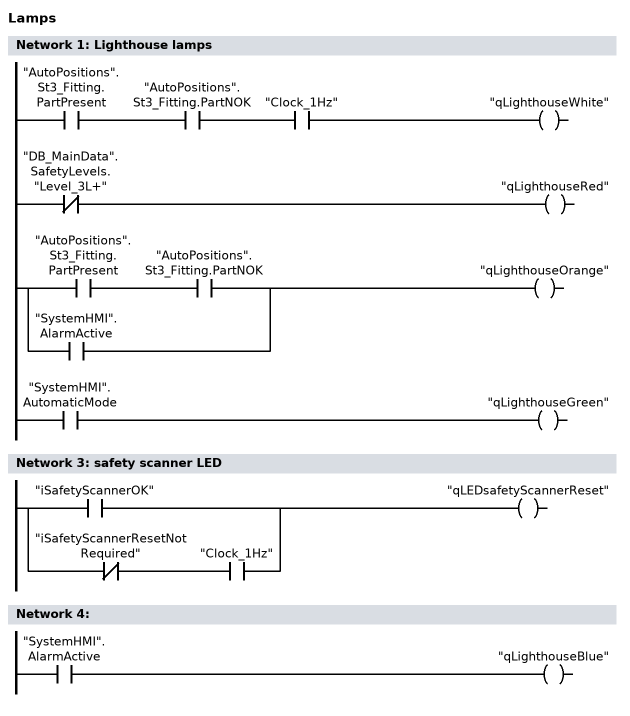
   RUNG wire#powerrail
      Contact( "AutoPositions".St3_Fitting.PartPresent )
      Contact( "AutoPositions".St3_Fitting.PartNOK )
      Contact( "Clock_1Hz" )
      Coil( "qLighthouseWhite" )
   END_RUNG
   RUNG wire#powerrail
      I_Contact( "DB_MainData".SafetyLevels."Level_3L+" )
      Coil( "qLighthouseRed" )
   END_RUNG
   RUNG wire#powerrail
      Contact( "AutoPositions".St3_Fitting.PartPresent )
      Contact( "AutoPositions".St3_Fitting.PartNOK )
      wire#w1
      Coil( "qLighthouseOrange" )
   END_RUNG
   RUNG wire#powerrail
      Contact( "SystemHMI".AlarmActive )
   END_RUNG wire#w1
   RUNG wire#powerrail
      Contact( "SystemHMI".AutomaticMode )
      Coil( "qLighthouseGreen" )
   END_RUNG
   // the same network as SCL:
   "qLighthouseWhite" := "AutoPositions".St3_Fitting.PartPresent AND "AutoPositions".St3_Fitting.PartNOK AND "Clock_1Hz";
   "qLighthouseRed" := NOT "DB_MainData".SafetyLevels."Level_3L+";
   "qLighthouseOrange" := ("AutoPositions".St3_Fitting.PartPresent AND "AutoPositions".St3_Fitting.PartNOK) OR "SystemHMI".AlarmActive;
   "qLighthouseGreen" := "SystemHMI".AutomaticMode;
END_REGION

REGION Network 2 (SCL): Alarm LED on OP
   //red button hmi
   "qResetAlarm" := "SystemHMI".AlarmActiveBlinking  AND "Clock_1Hz";
END_REGION

REGION Network 3: safety scanner LED
   RUNG wire#powerrail
      Contact( "iSafetyScannerOK" )
      wire#w1
      Coil( "qLEDsafetyScannerReset" )
   END_RUNG
   RUNG wire#powerrail
      I_Contact( "iSafetyScannerResetNotRequired" )
      Contact( "Clock_1Hz" )
   END_RUNG wire#w1
   // the same network as SCL:
   "qLEDsafetyScannerReset" := "iSafetyScannerOK" OR (NOT "iSafetyScannerResetNotRequired" AND "Clock_1Hz");
END_REGION

REGION Network 4
   RUNG wire#powerrail
      Contact( "SystemHMI".AlarmActive )
      Coil( "qLighthouseBlue" )
   END_RUNG
   // the same network as SCL:
   "qLighthouseBlue" := "SystemHMI".AlarmActive;
END_REGION
END_FUNCTION_BLOCK

FUNCTION_BLOCK "SandBox"
{ S7_Optimized_Access := 'TRUE' }
VERSION : 0.1

BEGIN
	;
END_FUNCTION_BLOCK

FUNCTION "Collisions" : Void
{ S7_Optimized_Access := 'TRUE' }
VERSION : 0.1

BEGIN
	;
	
	
END_FUNCTION

FUNCTION "READERS" : Void   // FC19, LAD
{ S7_Optimized_Access := 'TRUE' }
VERSION : 0.1
// stored: AutoNumber true, IsIECCheckEnabled false, SetENOAutomatically false, UDAEnableTagReadback false
   VAR_TEMP
      done1 : Bool;
      done2 : Bool;
      done3 : Bool;
      done4 : Bool;
      ERROR_RECIBIDO_ESCANER_REAR_TUBE : Int;
      ERROR_RECIBIDO_ESCANER_FRONT_TUBE : Int;
      ERROR_RECIBIDO_ESCANER_LH_MEMBER : Int;
      ERROR_RECIBIDO_ESCANER_RH_MEMBER : Int;
   END_VAR
   VAR_TEMP   // added for the SCL form of the ladder/FBD networks
      _w1 : Bool;
   END_VAR
BEGIN

REGION Network 1: INIT
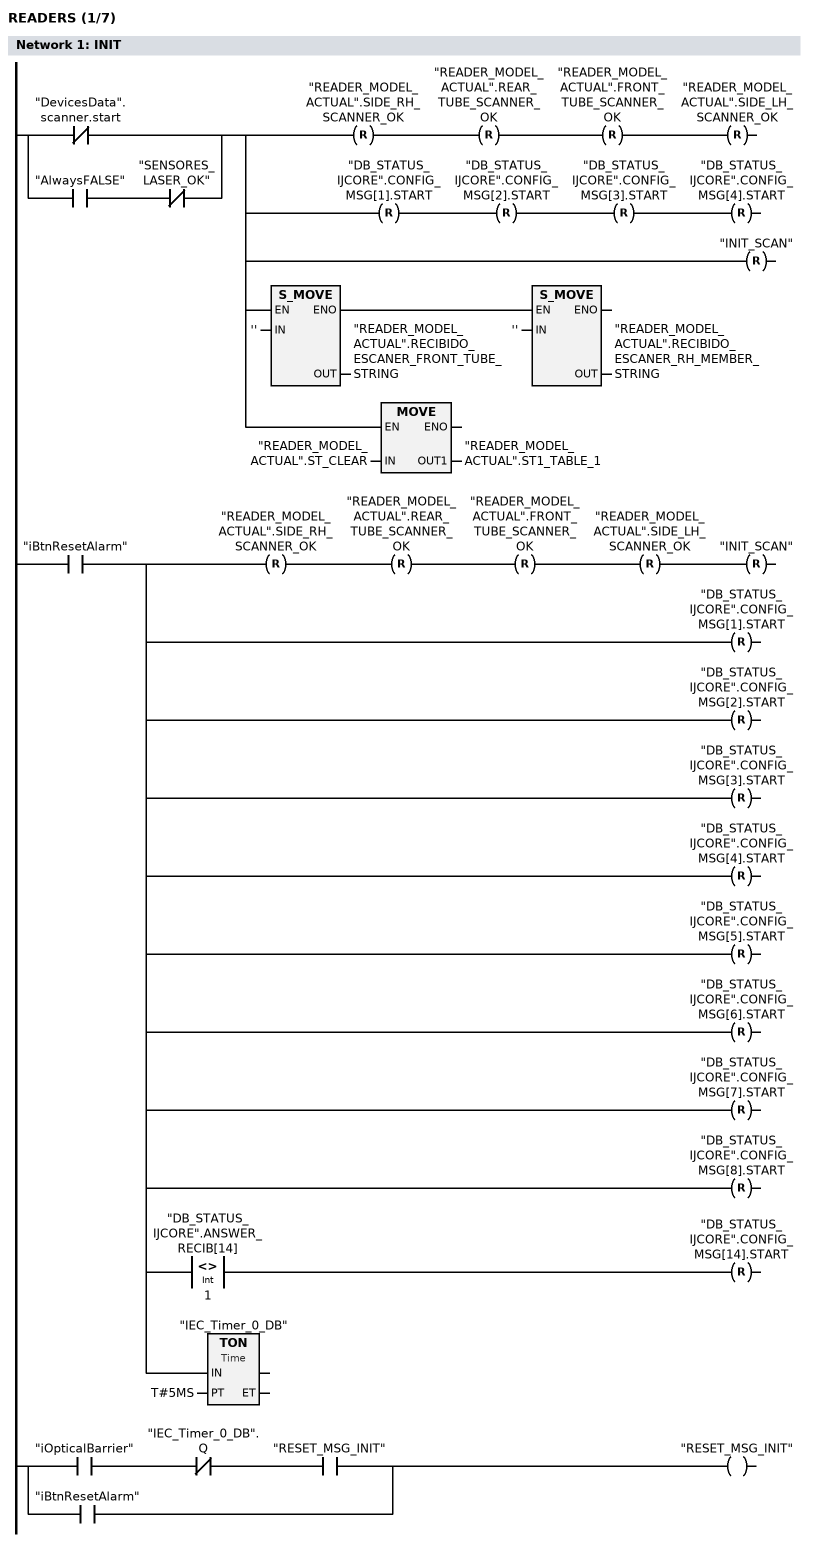
   RUNG wire#powerrail
      I_Contact( "DevicesData".scanner.start )
      wire#w1
      R_Coil( "READER_MODEL_ACTUAL".SIDE_RH_SCANNER_OK )
      R_Coil( "READER_MODEL_ACTUAL".REAR_TUBE_SCANNER_OK )
      R_Coil( "READER_MODEL_ACTUAL".FRONT_TUBE_SCANNER_OK )
      R_Coil( "READER_MODEL_ACTUAL".SIDE_LH_SCANNER_OK )
   END_RUNG
   RUNG wire#powerrail
      Contact( "AlwaysFALSE" )
      I_Contact( "SENSORES_LASER_OK" )
   END_RUNG wire#w1
   RUNG wire#w1
      R_Coil( "DB_STATUS_IJCORE".CONFIG_MSG[1].START )
      R_Coil( "DB_STATUS_IJCORE".CONFIG_MSG[2].START )
      R_Coil( "DB_STATUS_IJCORE".CONFIG_MSG[3].START )
      R_Coil( "DB_STATUS_IJCORE".CONFIG_MSG[4].START )
   END_RUNG
   RUNG wire#w1
      R_Coil( "INIT_SCAN" )
   END_RUNG
   RUNG wire#w1
      S_Move(in := '', out => "READER_MODEL_ACTUAL".RECIBIDO_ESCANER_FRONT_TUBE_STRING)
      S_Move(in := '', out => "READER_MODEL_ACTUAL".RECIBIDO_ESCANER_RH_MEMBER_STRING)
   END_RUNG
   RUNG wire#w1
      Move(in := "READER_MODEL_ACTUAL".ST_CLEAR, out1 => "READER_MODEL_ACTUAL".ST1_TABLE_1)
   END_RUNG
   RUNG wire#powerrail
      Contact( "iBtnResetAlarm" )
      wire#w2
      R_Coil( "READER_MODEL_ACTUAL".SIDE_RH_SCANNER_OK )
      R_Coil( "READER_MODEL_ACTUAL".REAR_TUBE_SCANNER_OK )
      R_Coil( "READER_MODEL_ACTUAL".FRONT_TUBE_SCANNER_OK )
      R_Coil( "READER_MODEL_ACTUAL".SIDE_LH_SCANNER_OK )
      R_Coil( "INIT_SCAN" )
   END_RUNG
   RUNG wire#w2
      R_Coil( "DB_STATUS_IJCORE".CONFIG_MSG[1].START )
   END_RUNG
   RUNG wire#w2
      R_Coil( "DB_STATUS_IJCORE".CONFIG_MSG[2].START )
   END_RUNG
   RUNG wire#w2
      R_Coil( "DB_STATUS_IJCORE".CONFIG_MSG[3].START )
   END_RUNG
   RUNG wire#w2
      R_Coil( "DB_STATUS_IJCORE".CONFIG_MSG[4].START )
   END_RUNG
   RUNG wire#w2
      R_Coil( "DB_STATUS_IJCORE".CONFIG_MSG[5].START )
   END_RUNG
   RUNG wire#w2
      R_Coil( "DB_STATUS_IJCORE".CONFIG_MSG[6].START )
   END_RUNG
   RUNG wire#w2
      R_Coil( "DB_STATUS_IJCORE".CONFIG_MSG[7].START )
   END_RUNG
   RUNG wire#w2
      R_Coil( "DB_STATUS_IJCORE".CONFIG_MSG[8].START )
   END_RUNG
   RUNG wire#w2
      { S7_Templates := "SrcType := Int" } NE_Contact(in1 := "DB_STATUS_IJCORE".ANSWER_RECIB[14], in2 := 1)
      R_Coil( "DB_STATUS_IJCORE".CONFIG_MSG[14].START )
   END_RUNG
   RUNG wire#w2
      { S7_Templates := "time_type := Time" } "IEC_Timer_0_DB".TON(pt := T#5MS, et =>)
   END_RUNG
   RUNG wire#powerrail
      Contact( "iOpticalBarrier" )
      I_Contact( "IEC_Timer_0_DB".Q )
      Contact( "RESET_MSG_INIT" )
      wire#w3
      Coil( "RESET_MSG_INIT" )
   END_RUNG
   RUNG wire#powerrail
      Contact( "iBtnResetAlarm" )
   END_RUNG wire#w3
   // the same network as SCL:
   IF NOT "DevicesData".scanner.start OR ("AlwaysFALSE" AND NOT "SENSORES_LASER_OK") THEN
       "READER_MODEL_ACTUAL".SIDE_RH_SCANNER_OK := FALSE;
       "READER_MODEL_ACTUAL".REAR_TUBE_SCANNER_OK := FALSE;
       "READER_MODEL_ACTUAL".FRONT_TUBE_SCANNER_OK := FALSE;
       "READER_MODEL_ACTUAL".SIDE_LH_SCANNER_OK := FALSE;
       "DB_STATUS_IJCORE".CONFIG_MSG[1].START := FALSE;
       "DB_STATUS_IJCORE".CONFIG_MSG[2].START := FALSE;
       "DB_STATUS_IJCORE".CONFIG_MSG[3].START := FALSE;
       "DB_STATUS_IJCORE".CONFIG_MSG[4].START := FALSE;
       "INIT_SCAN" := FALSE;
       "READER_MODEL_ACTUAL".RECIBIDO_ESCANER_FRONT_TUBE_STRING := '';
       "READER_MODEL_ACTUAL".RECIBIDO_ESCANER_RH_MEMBER_STRING := '';
       "READER_MODEL_ACTUAL".ST1_TABLE_1 := "READER_MODEL_ACTUAL".ST_CLEAR;
   END_IF;
   IF "iBtnResetAlarm" THEN
       "READER_MODEL_ACTUAL".SIDE_RH_SCANNER_OK := FALSE;
       "READER_MODEL_ACTUAL".REAR_TUBE_SCANNER_OK := FALSE;
       "READER_MODEL_ACTUAL".FRONT_TUBE_SCANNER_OK := FALSE;
       "READER_MODEL_ACTUAL".SIDE_LH_SCANNER_OK := FALSE;
       "INIT_SCAN" := FALSE;
       "DB_STATUS_IJCORE".CONFIG_MSG[1].START := FALSE;
       "DB_STATUS_IJCORE".CONFIG_MSG[2].START := FALSE;
       "DB_STATUS_IJCORE".CONFIG_MSG[3].START := FALSE;
       "DB_STATUS_IJCORE".CONFIG_MSG[4].START := FALSE;
       "DB_STATUS_IJCORE".CONFIG_MSG[5].START := FALSE;
       "DB_STATUS_IJCORE".CONFIG_MSG[6].START := FALSE;
       "DB_STATUS_IJCORE".CONFIG_MSG[7].START := FALSE;
       "DB_STATUS_IJCORE".CONFIG_MSG[8].START := FALSE;
   END_IF;
   IF "iBtnResetAlarm" AND ("DB_STATUS_IJCORE".ANSWER_RECIB[14] <> 1) THEN
       "DB_STATUS_IJCORE".CONFIG_MSG[14].START := FALSE;
   END_IF;
   "IEC_Timer_0_DB".TON(IN := "iBtnResetAlarm", PT := T#5MS);
   "RESET_MSG_INIT" := ("iOpticalBarrier" AND NOT "IEC_Timer_0_DB".Q AND "RESET_MSG_INIT") OR "iBtnResetAlarm";
END_REGION

REGION Network 2: CHARGE DATA FOR MODEL
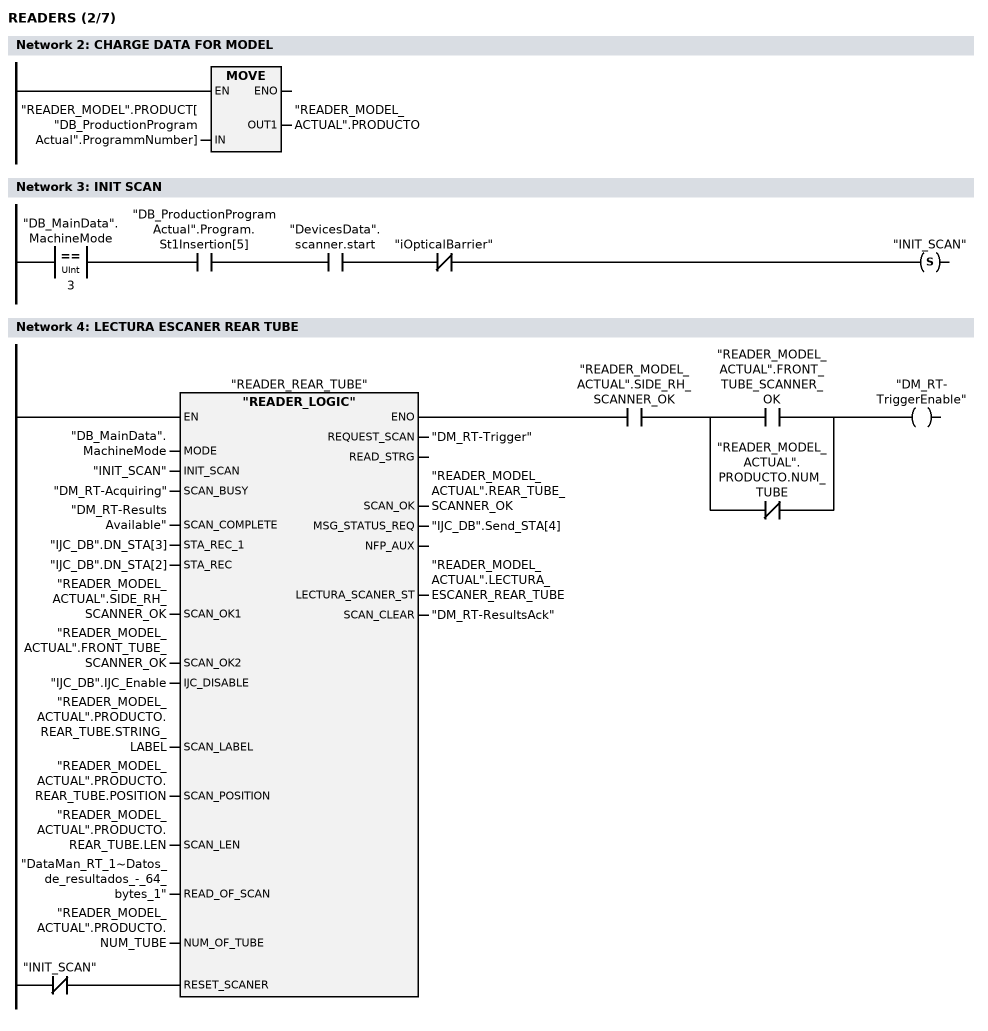
   RUNG wire#powerrail
      Move(in := "READER_MODEL".PRODUCT["DB_ProductionProgramActual".ProgrammNumber], out1 => "READER_MODEL_ACTUAL".PRODUCTO)
   END_RUNG
   // the same network as SCL:
   "READER_MODEL_ACTUAL".PRODUCTO := "READER_MODEL".PRODUCT["DB_ProductionProgramActual".ProgrammNumber];
END_REGION

REGION Network 3: INIT SCAN
   RUNG wire#powerrail
      { S7_Templates := "SrcType := UInt" } EQ_Contact(in1 := "DB_MainData".MachineMode, in2 := 3)
      Contact( "DB_ProductionProgramActual".Program.St1Insertion[5] )
      Contact( "DevicesData".scanner.start )
      I_Contact( "iOpticalBarrier" )
      S_Coil( "INIT_SCAN" )
   END_RUNG
   // the same network as SCL:
   IF ("DB_MainData".MachineMode = 3) AND "DB_ProductionProgramActual".Program.St1Insertion[5] AND "DevicesData".scanner.start AND NOT "iOpticalBarrier" THEN
       "INIT_SCAN" := TRUE;
   END_IF;
END_REGION

REGION Network 4: LECTURA ESCANER REAR TUBE
   RUNG wire#powerrail
      "READER_REAR_TUBE"(RESET_SCANER := wire#w1, MODE := "DB_MainData".MachineMode, INIT_SCAN := "INIT_SCAN", SCAN_BUSY := "DM_RT-Acquiring", SCAN_COMPLETE := "DM_RT-Results Available", STA_REC_1 := "IJC_DB".DN_STA[3], STA_REC := "IJC_DB".DN_STA[2], SCAN_OK1 := "READER_MODEL_ACTUAL".SIDE_RH_SCANNER_OK, SCAN_OK2 := "READER_MODEL_ACTUAL".FRONT_TUBE_SCANNER_OK, IJC_DISABLE := "IJC_DB".IJC_Enable, SCAN_LABEL := "READER_MODEL_ACTUAL".PRODUCTO.REAR_TUBE.STRING_LABEL, SCAN_POSITION := "READER_MODEL_ACTUAL".PRODUCTO.REAR_TUBE.POSITION, SCAN_LEN := "READER_MODEL_ACTUAL".PRODUCTO.REAR_TUBE.LEN, READ_OF_SCAN := "DataMan_RT_1~Datos_de_resultados_-_64_bytes_1", NUM_OF_TUBE := "READER_MODEL_ACTUAL".PRODUCTO.NUM_TUBE, REQUEST_SCAN => "DM_RT-Trigger", READ_STRG =>, SCAN_OK => "READER_MODEL_ACTUAL".REAR_TUBE_SCANNER_OK, MSG_STATUS_REQ => "IJC_DB".Send_STA[4], NFP_AUX =>, LECTURA_SCANER_ST => "READER_MODEL_ACTUAL".LECTURA_ESCANER_REAR_TUBE, SCAN_CLEAR => "DM_RT-ResultsAck")
      Contact( "READER_MODEL_ACTUAL".SIDE_RH_SCANNER_OK )
      wire#w2
      Contact( "READER_MODEL_ACTUAL".FRONT_TUBE_SCANNER_OK )
      wire#w3
      Coil( "DM_RT-TriggerEnable" )
   END_RUNG
   RUNG wire#powerrail
      I_Contact( "INIT_SCAN" )
   END_RUNG wire#w1
   RUNG wire#w2
      I_Contact( "READER_MODEL_ACTUAL".PRODUCTO.NUM_TUBE )
   END_RUNG wire#w3
   // the same network as SCL:
   "READER_REAR_TUBE"(MODE := "DB_MainData".MachineMode,   // "READER_LOGIC"
                      INIT_SCAN := "INIT_SCAN",
                      SCAN_BUSY := "DM_RT-Acquiring",
                      SCAN_COMPLETE := "DM_RT-Results Available",
                      STA_REC_1 := "IJC_DB".DN_STA[3],
                      STA_REC := "IJC_DB".DN_STA[2],
                      SCAN_OK1 := "READER_MODEL_ACTUAL".SIDE_RH_SCANNER_OK,
                      SCAN_OK2 := "READER_MODEL_ACTUAL".FRONT_TUBE_SCANNER_OK,
                      IJC_DISABLE := "IJC_DB".IJC_Enable,
                      SCAN_LABEL := "READER_MODEL_ACTUAL".PRODUCTO.REAR_TUBE.STRING_LABEL,
                      SCAN_POSITION := "READER_MODEL_ACTUAL".PRODUCTO.REAR_TUBE.POSITION,
                      SCAN_LEN := "READER_MODEL_ACTUAL".PRODUCTO.REAR_TUBE.LEN,
                      READ_OF_SCAN := "DataMan_RT_1~Datos_de_resultados_-_64_bytes_1",
                      NUM_OF_TUBE := "READER_MODEL_ACTUAL".PRODUCTO.NUM_TUBE,
                      RESET_SCANER := NOT "INIT_SCAN",
                      REQUEST_SCAN => "DM_RT-Trigger",
                      SCAN_OK => "READER_MODEL_ACTUAL".REAR_TUBE_SCANNER_OK,
                      MSG_STATUS_REQ => "IJC_DB".Send_STA[4],
                      LECTURA_SCANER_ST => "READER_MODEL_ACTUAL".LECTURA_ESCANER_REAR_TUBE,
                      SCAN_CLEAR => "DM_RT-ResultsAck",
                      ENO => #_w1);
   "DM_RT-TriggerEnable" := #_w1 AND "READER_MODEL_ACTUAL".SIDE_RH_SCANNER_OK AND ("READER_MODEL_ACTUAL".FRONT_TUBE_SCANNER_OK OR NOT "READER_MODEL_ACTUAL".PRODUCTO.NUM_TUBE);
END_REGION

REGION Network 5: LECTURA ESCANER FRONT TUBE
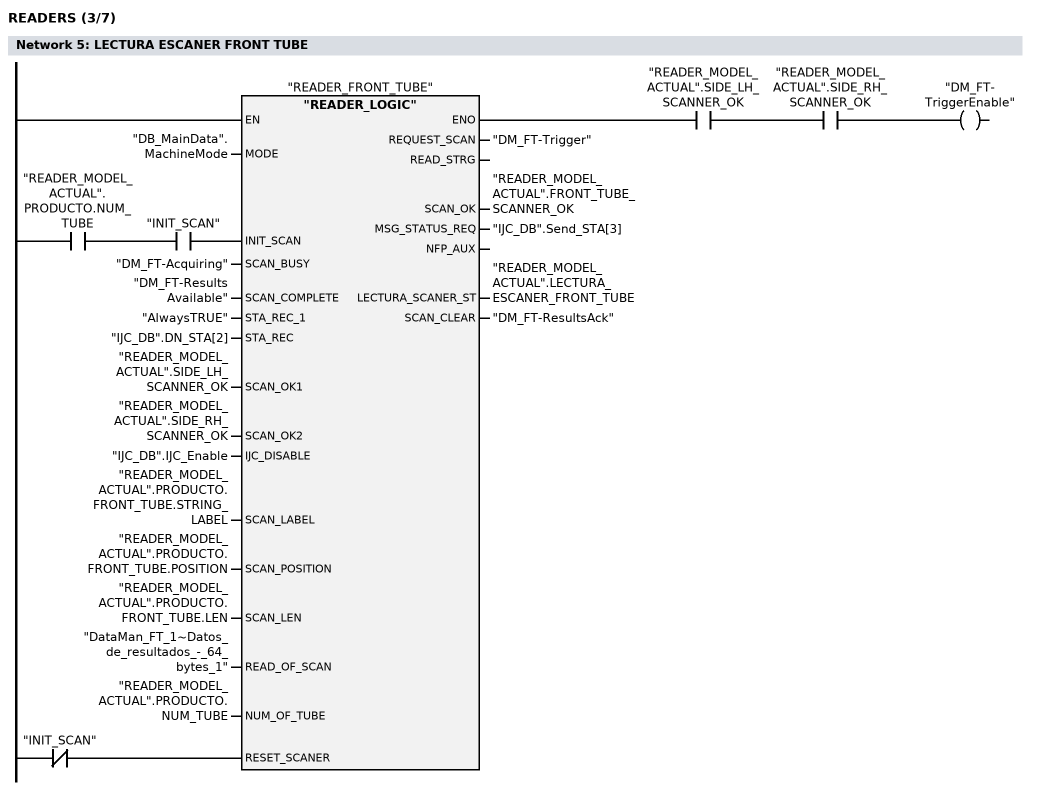
   RUNG wire#powerrail
      "READER_FRONT_TUBE"(INIT_SCAN := wire#w1, RESET_SCANER := wire#w2, MODE := "DB_MainData".MachineMode, SCAN_BUSY := "DM_FT-Acquiring", SCAN_COMPLETE := "DM_FT-Results Available", STA_REC_1 := "AlwaysTRUE", STA_REC := "IJC_DB".DN_STA[2], SCAN_OK1 := "READER_MODEL_ACTUAL".SIDE_LH_SCANNER_OK, SCAN_OK2 := "READER_MODEL_ACTUAL".SIDE_RH_SCANNER_OK, IJC_DISABLE := "IJC_DB".IJC_Enable, SCAN_LABEL := "READER_MODEL_ACTUAL".PRODUCTO.FRONT_TUBE.STRING_LABEL, SCAN_POSITION := "READER_MODEL_ACTUAL".PRODUCTO.FRONT_TUBE.POSITION, SCAN_LEN := "READER_MODEL_ACTUAL".PRODUCTO.FRONT_TUBE.LEN, READ_OF_SCAN := "DataMan_FT_1~Datos_de_resultados_-_64_bytes_1", NUM_OF_TUBE := "READER_MODEL_ACTUAL".PRODUCTO.NUM_TUBE, REQUEST_SCAN => "DM_FT-Trigger", READ_STRG =>, SCAN_OK => "READER_MODEL_ACTUAL".FRONT_TUBE_SCANNER_OK, MSG_STATUS_REQ => "IJC_DB".Send_STA[3], NFP_AUX =>, LECTURA_SCANER_ST => "READER_MODEL_ACTUAL".LECTURA_ESCANER_FRONT_TUBE, SCAN_CLEAR => "DM_FT-ResultsAck")
      Contact( "READER_MODEL_ACTUAL".SIDE_LH_SCANNER_OK )
      Contact( "READER_MODEL_ACTUAL".SIDE_RH_SCANNER_OK )
      Coil( "DM_FT-TriggerEnable" )
   END_RUNG
   RUNG wire#powerrail
      Contact( "READER_MODEL_ACTUAL".PRODUCTO.NUM_TUBE )
      Contact( "INIT_SCAN" )
   END_RUNG wire#w1
   RUNG wire#powerrail
      I_Contact( "INIT_SCAN" )
   END_RUNG wire#w2
   // the same network as SCL:
   "READER_FRONT_TUBE"(MODE := "DB_MainData".MachineMode,   // "READER_LOGIC"
                       INIT_SCAN := "READER_MODEL_ACTUAL".PRODUCTO.NUM_TUBE AND "INIT_SCAN",
                       SCAN_BUSY := "DM_FT-Acquiring",
                       SCAN_COMPLETE := "DM_FT-Results Available",
                       STA_REC_1 := "AlwaysTRUE",
                       STA_REC := "IJC_DB".DN_STA[2],
                       SCAN_OK1 := "READER_MODEL_ACTUAL".SIDE_LH_SCANNER_OK,
                       SCAN_OK2 := "READER_MODEL_ACTUAL".SIDE_RH_SCANNER_OK,
                       IJC_DISABLE := "IJC_DB".IJC_Enable,
                       SCAN_LABEL := "READER_MODEL_ACTUAL".PRODUCTO.FRONT_TUBE.STRING_LABEL,
                       SCAN_POSITION := "READER_MODEL_ACTUAL".PRODUCTO.FRONT_TUBE.POSITION,
                       SCAN_LEN := "READER_MODEL_ACTUAL".PRODUCTO.FRONT_TUBE.LEN,
                       READ_OF_SCAN := "DataMan_FT_1~Datos_de_resultados_-_64_bytes_1",
                       NUM_OF_TUBE := "READER_MODEL_ACTUAL".PRODUCTO.NUM_TUBE,
                       RESET_SCANER := NOT "INIT_SCAN",
                       REQUEST_SCAN => "DM_FT-Trigger",
                       SCAN_OK => "READER_MODEL_ACTUAL".FRONT_TUBE_SCANNER_OK,
                       MSG_STATUS_REQ => "IJC_DB".Send_STA[3],
                       LECTURA_SCANER_ST => "READER_MODEL_ACTUAL".LECTURA_ESCANER_FRONT_TUBE,
                       SCAN_CLEAR => "DM_FT-ResultsAck",
                       ENO => #_w1);
   "DM_FT-TriggerEnable" := #_w1 AND "READER_MODEL_ACTUAL".SIDE_LH_SCANNER_OK AND "READER_MODEL_ACTUAL".SIDE_RH_SCANNER_OK;
END_REGION

